        (* Warnung Hand Ein *)
		ayWarningReporter[3].proPrio	:= 3;    
		ayWarningReporter[3].proHandLokal :=    xIsHandOn;
		ayWarningReporter[3].metReport(			xSetReportIn					:= xIsHandOn,
												iReportID						:= 3,
												enReportTypeIn					:= CtaAppReport.enReportType.Warning,  
												enReportAcknowledgeTypeIn   	:= CtaAppReport.enReportAcknowledgeType.Auto,
												tDelay							:= T#0S, 
												ITF_BMK_IN						:= THIS^,			              
												pstReportTextListIn				:= ADR(GlobalKonstant.stReportTextListWarning),
												stOptionalReportText		    := '',   
												iRetryTilReportLock 		    := 0, 
												xResetCount         		    := FALSE,  
												tReset						    := T#0S);   
 
        (* Warnung Handmodul Actuator *)
		ayWarningReporter[4].proPrio	:= 4;    
		ayWarningReporter[4].proHandLokal :=    xActuatorHand;
		ayWarningReporter[4].metReport(			xSetReportIn					:= xActuatorHand,
												iReportID						:= 4,
												enReportTypeIn					:= CtaAppReport.enReportType.Warning,  
												enReportAcknowledgeTypeIn   	:= CtaAppReport.enReportAcknowledgeType.Auto,
												tDelay							:= T#0S, 
												ITF_BMK_IN						:= THIS^,			              
												pstReportTextListIn				:= ADR(GlobalKonstant.stReportTextListWarning),
												stOptionalReportText		    := '',   
												iRetryTilReportLock 		    := 0, 
												xResetCount         		    := FALSE,  
												tReset						    := T#0S);                                                   
(* Sync Reports *)                                         
FOR difor := LOWER_BOUND(ayErrorReporter,1) TO UPPER_BOUND(ayErrorReporter,1) DO
	fbReportManager.metSyncReporter(ayErrorReporter[difor]);	
END_FOR;
FOR difor := LOWER_BOUND(ayWarningReporter,1) TO UPPER_BOUND(ayWarningReporter,1) DO
	fbReportManager.metSyncReporter(ayWarningReporter[difor]);	
END_FOR;
                                                                             
_xIsError   := scEWI.iError <> 0;
_xIsWarning := scEWI.iWarning <> 0;
END_ACTION

{attribute 'monitoring' := 'variable'}
PROPERTY proAcknowlege : BOOL
GET
proAcknowlege :=NOT proIsError;
END_GET
END_PROPERTY

{attribute 'monitoring' := 'variable'}
PROPERTY proAvailable : BOOL
GET
proAvailable := proIsReady;
END_GET
END_PROPERTY

{attribute 'monitoring' := 'variable'}
PROPERTY proLockDown : BOOL
GET
proLockDown := proIsError;
END_GET
END_PROPERTY

END_FUNCTION_BLOCK

// 30 Program Organization Units/Abstracte Bausteine/fbSperrAntriebTabellenInfo
{attribute 'hide'} 
FUNCTION_BLOCK INTERNAL ABSTRACT fbSperrAntriebTabellenInfo EXTENDS CtaAppBmk.fbBMK IMPLEMENTS ITF_SPERRANTRIEB_TABELLE_INFO

PROPERTY proOnAuf : BOOL
GET
END_GET
END_PROPERTY

PROPERTY proStateSymbol : STRING
GET
END_GET
END_PROPERTY

PROPERTY proEnSymbol : STRING
GET
END_GET
END_PROPERTY

PROPERTY proIsOn : BOOL
GET
END_GET
END_PROPERTY

PROPERTY proIsOnY : REAL
GET
END_GET
END_PROPERTY

PROPERTY proOn : BOOL
GET
END_GET
END_PROPERTY

PROPERTY proOnY : REAL
GET
END_GET
END_PROPERTY

PROPERTY proOnZu : BOOL
GET
END_GET
END_PROPERTY

PROPERTY proRükIsClosed : BOOL
GET
END_GET
END_PROPERTY

PROPERTY proRükIsOpen : BOOL
GET
END_GET
END_PROPERTY

END_FUNCTION_BLOCK

// 21 Interface/ITF_SPERRANTRIEB_TABELLE_INFO
INTERFACE INTERNAL ITF_SPERRANTRIEB_TABELLE_INFO EXTENDS CtaAppBmk.ITF_BMK

PROPERTY proRükIsOpen : BOOL
GET
END_GET
END_PROPERTY

PROPERTY proRükIsClosed : BOOL
GET
END_GET
END_PROPERTY

PROPERTY INTERNAL proStateSymbol : STRING
GET
END_GET
END_PROPERTY

PROPERTY INTERNAL proEnSymbol : STRING
GET
END_GET
END_PROPERTY

PROPERTY proOnZu : BOOL
GET
END_GET
END_PROPERTY

PROPERTY proIsOnY : REAL
GET
END_GET
END_PROPERTY

PROPERTY proOnAuf : BOOL
GET
END_GET
END_PROPERTY

PROPERTY proOnY : REAL
GET
END_GET
END_PROPERTY

END_INTERFACE

// 21 Interface/ITF_SPERRANTRIEB
INTERFACE ITF_SPERRANTRIEB EXTENDS ITF_SPERRANTRIEB_TABELLE_INFO, CtaAppModbusSpezifikation.ITF_MODBUS_SPEZIFIKATION

PROPERTY proAuto : BOOL
GET
END_GET
SET
END_SET
END_PROPERTY

PROPERTY proHandOff : BOOL
GET
END_GET
SET
END_SET
END_PROPERTY

PROPERTY proHandOn : BOOL
GET
END_GET
SET
END_SET
END_PROPERTY

PROPERTY proIsRegulatet : BOOL
GET
END_GET
END_PROPERTY

PROPERTY proIsError : BOOL
GET
END_GET
END_PROPERTY

PROPERTY proIsWarning : BOOL
GET
END_GET
END_PROPERTY

PROPERTY proIsEnabled : BOOL
GET
END_GET
END_PROPERTY

PROPERTY proIsHandOnOrOff : BOOL
GET
END_GET
END_PROPERTY

PROPERTY proIsReady : BOOL
GET
END_GET
END_PROPERTY

PROPERTY proHardWareHandModulAktive : BOOL
GET
END_GET
END_PROPERTY

PROPERTY proRevisionSwitchOk : BOOL
GET
END_GET
END_PROPERTY

PROPERTY proHandManualClose : BOOL
SET
END_SET
GET
END_GET
END_PROPERTY

PROPERTY proEn : BOOL
SET
END_SET
GET
END_GET
END_PROPERTY

PROPERTY proGetDI_RükIsOpen : BOOL
GET
END_GET
END_PROPERTY

PROPERTY proNotShowDI_RükIsOpen : BOOL
GET
END_GET
END_PROPERTY

PROPERTY proIsOpen_ITF : CtaSysIO.ITF_IO
GET
END_GET
END_PROPERTY

PROPERTY INTERNAL proGetDI_ActuatorHand : BOOL
GET
END_GET
END_PROPERTY

PROPERTY proNotShowDI_ActuatorHand : BOOL
GET
END_GET
END_PROPERTY

PROPERTY proHandModul_ITF : CtaSysIO.ITF_IO
GET
END_GET
END_PROPERTY

PROPERTY INTERNAL proGetDI_ActuatorFuseOk : BOOL
GET
END_GET
END_PROPERTY

PROPERTY proNotShowDI_ActuatorFuseOk : BOOL
GET
END_GET
END_PROPERTY

PROPERTY proActuatorFuse_ITF : CtaSysIO.ITF_IO
GET
END_GET
END_PROPERTY

PROPERTY INTERNAL proGetDI_IsReady : BOOL
GET
END_GET
END_PROPERTY

PROPERTY proNotShowDI_Ready : BOOL
GET
END_GET
END_PROPERTY

PROPERTY proActuatorReady_ITF : CtaSysIO.ITF_IO
GET
END_GET
END_PROPERTY

PROPERTY INTERNAL proGetDI_FuseOK : BOOL
GET
END_GET
END_PROPERTY

PROPERTY proNotShowDI_FuseOk : BOOL
GET
END_GET
END_PROPERTY

PROPERTY proFuse_ITF : CtaSysIO.ITF_IO
GET
END_GET
END_PROPERTY

PROPERTY INTERNAL proGetDI_RevisionSwitchOK : BOOL
GET
END_GET
END_PROPERTY

PROPERTY proNotShowDI_RevisionSwitchOk : BOOL
GET
END_GET
END_PROPERTY

PROPERTY proRevisionSwitch_ITF : CtaSysIO.ITF_IO
GET
END_GET
END_PROPERTY

PROPERTY proNotShowAI_ActualPosition : BOOL
GET
END_GET
END_PROPERTY

PROPERTY proGetAI_ActualPosition : REAL
GET
END_GET
END_PROPERTY

PROPERTY proActualPosition_ITF : CtaSysIO.ITF_IO
GET
END_GET
END_PROPERTY

PROPERTY proGetDI_RükIsClosed : BOOL
GET
END_GET
END_PROPERTY

PROPERTY proNotShowDI_RükIsClosed : BOOL
GET
END_GET
END_PROPERTY

PROPERTY proIsClosed_ITF : CtaSysIO.ITF_IO
GET
END_GET
END_PROPERTY

PROPERTY proOnY_ITF : CtaSysIO.ITF_IO
GET
END_GET
END_PROPERTY

PROPERTY proOnOpen_ITF : CtaSysIO.ITF_IO
GET
END_GET
END_PROPERTY

PROPERTY proOnClose_ITF : CtaSysIO.ITF_IO
GET
END_GET
END_PROPERTY

PROPERTY INTERNAL proAnzWarning : INT
GET
END_GET
END_PROPERTY

PROPERTY INTERNAL proITF_REPORTMANAGER : CtaAppReport.ITF_REPORTMANAGER
GET
END_GET
END_PROPERTY

PROPERTY INTERNAL proAnzInfo : INT
GET
END_GET
END_PROPERTY

PROPERTY INTERNAL proAnzError : INT
GET
END_GET
END_PROPERTY

PROPERTY INTERNAL proModbusTest : BOOL
SET
END_SET
GET
END_GET
END_PROPERTY

PROPERTY proModbusStateWord : REFERENCE TO ARRAY[0..3] OF WORD
GET
END_GET
END_PROPERTY

PROPERTY proModbusControllWord : REFERENCE TO ARRAY[0..3] OF WORD
GET
END_GET
END_PROPERTY

PROPERTY proConfigError : BOOL
GET
END_GET
END_PROPERTY

PROPERTY p_scBase_fbxEnable : CtaSysConfig.ITF_DATATYPE;
GET
END_GET
END_PROPERTY

PROPERTY p_scBase_fbxControllMb : CtaSysConfig.ITF_DATATYPE;
GET
END_GET
END_PROPERTY

PROPERTY p_scBase_fbxInvertiert : CtaSysConfig.ITF_DATATYPE;
GET
END_GET
END_PROPERTY

PROPERTY p_scBase_fbtSettingTime : CtaSysConfig.ITF_DATATYPE;
GET
END_GET
END_PROPERTY

PROPERTY p_scFuse_fbxEnable : CtaSysConfig.ITF_DATATYPE;
GET
END_GET
END_PROPERTY

PROPERTY p_scFuse_fbxInputMb : CtaSysConfig.ITF_DATATYPE;
GET
END_GET
END_PROPERTY

PROPERTY p_scFuse_fbxDoesAlarm : CtaSysConfig.ITF_DATATYPE;
GET
END_GET
END_PROPERTY

PROPERTY p_scActuatorFuse_fbxEnable : CtaSysConfig.ITF_DATATYPE;
GET
END_GET
END_PROPERTY

PROPERTY p_scActuatorFuse_fbxInputMb : CtaSysConfig.ITF_DATATYPE;
GET
END_GET
END_PROPERTY

PROPERTY p_scActuatorFuse_fbxDoesAlarm : CtaSysConfig.ITF_DATATYPE;
GET
END_GET
END_PROPERTY

PROPERTY p_scInSperrAtRevisionSwitch_fbxEnable : CtaSysConfig.ITF_DATATYPE;
GET
END_GET
END_PROPERTY

PROPERTY p_scInSperrAtRevisionSwitch_fbxInputMb : CtaSysConfig.ITF_DATATYPE;
GET
END_GET
END_PROPERTY

PROPERTY p_scInSperrAtReady_fbxEnable : CtaSysConfig.ITF_DATATYPE;
GET
END_GET
END_PROPERTY

PROPERTY p_scInSperrAtReady_fbxInputMb : CtaSysConfig.ITF_DATATYPE;
GET
END_GET
END_PROPERTY

PROPERTY p_scInSperrAtHand_fbxEnable : CtaSysConfig.ITF_DATATYPE;
GET
END_GET
END_PROPERTY

PROPERTY p_scInSperrAtHand_fbxInputMb : CtaSysConfig.ITF_DATATYPE;
GET
END_GET
END_PROPERTY

PROPERTY p_scInSperrAtRükClosed_fbxEnable : CtaSysConfig.ITF_DATATYPE;
GET
END_GET
END_PROPERTY

PROPERTY p_scInSperrAtRükClosed_fbxInputMb : CtaSysConfig.ITF_DATATYPE;
GET
END_GET
END_PROPERTY

PROPERTY p_scInSperrAtRükClosed_fbxDoesAlarm : CtaSysConfig.ITF_DATATYPE;
GET
END_GET
END_PROPERTY

PROPERTY p_scInSperrAtRükClosed_fbtDelayStart : CtaSysConfig.ITF_DATATYPE;
GET
END_GET
END_PROPERTY

PROPERTY p_scInSperrAtRükClosed_fbtDelayRun : CtaSysConfig.ITF_DATATYPE;
GET
END_GET
END_PROPERTY

PROPERTY p_scInSperrAtRükClosed_fbiTypeOfAck : CtaSysConfig.ITF_DATATYPE;
GET
END_GET
END_PROPERTY

PROPERTY p_scInSperrAtRükClosed_fbiMaxErrorRetryAllowed : CtaSysConfig.ITF_DATATYPE;
GET
END_GET
END_PROPERTY

PROPERTY p_scInSperrAtRükOpen_fbxEnable : CtaSysConfig.ITF_DATATYPE;
GET
END_GET
END_PROPERTY

PROPERTY p_scInSperrAtRükOpen_fbxInputMb : CtaSysConfig.ITF_DATATYPE;
GET
END_GET
END_PROPERTY

PROPERTY p_scInSperrAtRükOpen_fbxDoesAlarm : CtaSysConfig.ITF_DATATYPE;
GET
END_GET
END_PROPERTY

PROPERTY p_scInSperrAtRükOpen_fbtDelayStart : CtaSysConfig.ITF_DATATYPE;
GET
END_GET
END_PROPERTY

PROPERTY p_scInSperrAtRükOpen_fbtDelayRun : CtaSysConfig.ITF_DATATYPE;
GET
END_GET
END_PROPERTY

PROPERTY p_scInSperrAtRükOpen_fbiTypeOfAck : CtaSysConfig.ITF_DATATYPE;
GET
END_GET
END_PROPERTY

PROPERTY p_scInSperrAtRükOpen_fbiMaxErrorRetryAllowed : CtaSysConfig.ITF_DATATYPE;
GET
END_GET
END_PROPERTY

PROPERTY p_scInSperrAtActualPosition_fbxEnable : CtaSysConfig.ITF_DATATYPE;
GET
END_GET
END_PROPERTY

PROPERTY p_scInSperrAtActualPosition_fbxInputMb : CtaSysConfig.ITF_DATATYPE;
GET
END_GET
END_PROPERTY

PROPERTY p_scInSperrAtActualPosition_fbxDoesAlarm : CtaSysConfig.ITF_DATATYPE;
GET
END_GET
END_PROPERTY

PROPERTY p_scInSperrAtActualPosition_fbrMaxDiff : CtaSysConfig.ITF_DATATYPE;
GET
END_GET
END_PROPERTY

PROPERTY p_scInSperrAtActualPosition_fbtDelayStart : CtaSysConfig.ITF_DATATYPE;
GET
END_GET
END_PROPERTY

PROPERTY p_scInSperrAtActualPosition_fbtDelayRun : CtaSysConfig.ITF_DATATYPE;
GET
END_GET
END_PROPERTY

PROPERTY p_scInSperrAtActualPosition_fbiTypeOfAck : CtaSysConfig.ITF_DATATYPE;
GET
END_GET
END_PROPERTY

PROPERTY p_scInSperrAtActualPosition_fbiMaxErrorRetryAllowed : CtaSysConfig.ITF_DATATYPE;
GET
END_GET
END_PROPERTY

PROPERTY p_scInfluxDb_fbxEnable : CtaSysConfig.ITF_DATATYPE;
GET
END_GET
END_PROPERTY

PROPERTY p_scManual_fbxAlowManualOn : CtaSysConfig.ITF_DATATYPE;
GET
END_GET
END_PROPERTY

PROPERTY p_scManual_fbuiManualState : CtaSysConfig.ITF_DATATYPE;
GET
END_GET
END_PROPERTY

PROPERTY p_scManual_fbuiSchaltBefehl : CtaSysConfig.ITF_DATATYPE;
GET
END_GET
END_PROPERTY

PROPERTY proHandManualOpen : BOOL
GET
END_GET
SET
END_SET
END_PROPERTY

PROPERTY proIsInverted : BOOL
GET
END_GET
END_PROPERTY

PROPERTY proKlappenStatus : enKlappenStatus
GET
END_GET
END_PROPERTY

PROPERTY proValveIcon : UINT
GET
END_GET
SET
END_SET
END_PROPERTY

{attribute 'monitoring' := 'variable'}
PROPERTY proAcknowlege : BOOL
GET
END_GET
END_PROPERTY

{attribute 'monitoring' := 'variable'}
PROPERTY proAvailable : BOOL
GET
END_GET
END_PROPERTY

{attribute 'monitoring' := 'variable'}
PROPERTY proLockDown : BOOL
GET
END_GET
END_PROPERTY

PROPERTY proOn : BOOL
GET
END_GET
END_PROPERTY

END_INTERFACE

// 30 Program Organization Units/fbSperrAntrieb_Collector
FUNCTION_BLOCK fbSperrAntrieb_Collector IMPLEMENTS ITF_SPERRAT_COLLECTOR
VAR_INPUT
END_VAR
VAR_OUTPUT
END_VAR
VAR
    aySperrAT_INTERFACE          : ARRAY[1..Parameter.iMaxSperrAntrieb] OF ITF_SPERRANTRIEB;   
    aySperrAT_INTERFACE_SORTET   : ARRAY[1..Parameter.iMaxSperrAntrieb] OF ITF_SPERRANTRIEB; 
    xIsSortet               : BOOL;
    diNext                  : DINT    := 1;
    diMin                   : DINT    := 1;
    diMax                   : DINT;
    diMaxSort               : DINT;
    xError                  : BOOL;
    xBufferError            : BOOL;
    diMissedBuffer          : DINT;
END_VAR

METHOD metRegistry : DINT
VAR_INPUT
    ITF_AT_IN   :   ITF_SPERRANTRIEB;
END_VAR
VAR
    diArrayPos  :   DINT;
    diCount     :   DINT;
END_VAR
IF ITF_AT_IN <> 0 THEN
    diArrayPos := __XADD(ADR(diNext),1);
    IF diArrayPos <= Parameter.iMaxSperrAntrieb AND diArrayPos >= 1 THEN
        IF __QUERYINTERFACE(ITF_AT_IN,aySperrAT_INTERFACE[diArrayPos]) THEN
            metRegistry             := diArrayPos;
            GVL_SperrAntrieb.xValidData       := TRUE;
            diCount    := __XADD(ADR(diMax),1);
        END_IF;
    ELSE
        IF diArrayPos > Parameter.iMaxSperrAntrieb THEN
            xBufferError := TRUE;
            diMissedBuffer := diArrayPos - Parameter.iMaxSperrAntrieb;
		END_IF;
        xError      := TRUE; 
        metRegistry := 0;
    END_IF;   
ELSE
    xError := TRUE; 
    metRegistry := 0;
END_IF;
END_METHOD

METHOD metSortArray
VAR_INPUT
    stSearch    :   STRING;
    uiSort      :   UINT;
END_VAR
VAR
    diFor1      :   DINT;
    diFor2      :   DINT;
    diFill      :   DINT;
    ITF_AT_Temp :   ITF_SPERRANTRIEB;    
    iBigger     :   INT;
END_VAR
IF stSearch <> '' THEN
    diMaxSort   := 0;
    diFill      := LOWER_BOUND(aySperrAT_INTERFACE,1); 
    FOR diFor1 := LOWER_BOUND(aySperrAT_INTERFACE,1) TO UPPER_BOUND(aySperrAT_INTERFACE,1) DO
        IF aySperrAT_INTERFACE[diFor1] <> 0 THEN
            IF FIND(aySperrAT_INTERFACE[diFor1].proGetBMK,stSearch) <> 0 OR FIND(aySperrAT_INTERFACE[diFor1].proGetVendorDesignation,stSearch) <> 0 THEN
                aySperrAT_INTERFACE_SORTET[diFill] := aySperrAT_INTERFACE[diFor1];
                diFill      := diFill + 1; 
                diMaxSort   := diFill -1; 
            END_IF;
        END_IF;
	END_FOR;
ELSE
    aySperrAT_INTERFACE_SORTET := aySperrAT_INTERFACE;
    diMaxSort := diMax;
END_IF; 
// 1 = Sort BMK
IF uiSort = 1 THEN
    FOR diFor1 := LOWER_BOUND(aySperrAT_INTERFACE_SORTET,1) TO diMaxSort DO 
        FOR diFor2 := LOWER_BOUND(aySperrAT_INTERFACE_SORTET,1) TO diMaxSort -1 DO 
            IF aySperrAT_INTERFACE_SORTET[diFor2] <> 0 AND aySperrAT_INTERFACE_SORTET[diFor2 + 1] <> 0 THEN
                IF LEN(aySperrAT_INTERFACE_SORTET[diFor2].proGetBMK) > LEN(aySperrAT_INTERFACE_SORTET[diFor2 + 1].proGetBMK) THEN
                    ITF_AT_Temp                         := aySperrAT_INTERFACE_SORTET[diFor2];
                    aySperrAT_INTERFACE_SORTET[diFor2]       := aySperrAT_INTERFACE_SORTET[diFor2 + 1];
                    aySperrAT_INTERFACE_SORTET[diFor2 + 1]   := ITF_AT_Temp; 
                ELSIF LEN(aySperrAT_INTERFACE_SORTET[diFor2].proGetBMK) = LEN(aySperrAT_INTERFACE_SORTET[diFor2 + 1].proGetBMK) THEN
                    iBigger := fcGetBigerStringValue(aySperrAT_INTERFACE_SORTET[diFor2].proGetBMK,aySperrAT_INTERFACE_SORTET[diFor2 + 1].proGetBMK);
                    IF iBigger = 1 THEN
                        ITF_AT_Temp                         := aySperrAT_INTERFACE_SORTET[diFor2];
                        aySperrAT_INTERFACE_SORTET[diFor2]       := aySperrAT_INTERFACE_SORTET[diFor2 + 1];
                        aySperrAT_INTERFACE_SORTET[diFor2 + 1]   := ITF_AT_Temp;                                                
					END_IF;
				END_IF;
            END_IF;       
        END_FOR;      
    END_FOR;     
// 2 = Sort Vendor Name    
ELSIF uiSort = 2 THEN
    FOR diFor1 := LOWER_BOUND(aySperrAT_INTERFACE_SORTET,1) TO diMaxSort DO 
        FOR diFor2 := LOWER_BOUND(aySperrAT_INTERFACE_SORTET,1) TO diMaxSort -1 DO 
            IF aySperrAT_INTERFACE_SORTET[diFor2] <> 0 AND aySperrAT_INTERFACE_SORTET[diFor2 + 1] <> 0 THEN
                iBigger := fcGetBigerStringValue(aySperrAT_INTERFACE_SORTET[diFor2].proGetVendorDesignation,aySperrAT_INTERFACE_SORTET[diFor2 + 1].proGetVendorDesignation);
                IF iBigger = 1 THEN
                    ITF_AT_Temp                         := aySperrAT_INTERFACE_SORTET[diFor2];
                    aySperrAT_INTERFACE_SORTET[diFor2]       := aySperrAT_INTERFACE_SORTET[diFor2 + 1];
                    aySperrAT_INTERFACE_SORTET[diFor2 + 1]   := ITF_AT_Temp;                                            
                END_IF;
            END_IF;       
        END_FOR;      
    END_FOR;
// 3 & 4 = Sort State  
ELSIF uiSort = 3 OR uiSort = 4 THEN
    FOR diFor1 := LOWER_BOUND(aySperrAT_INTERFACE_SORTET,1) TO diMaxSort DO 
        FOR diFor2 := LOWER_BOUND(aySperrAT_INTERFACE_SORTET,1) TO diMaxSort -1 DO 
            IF aySperrAT_INTERFACE_SORTET[diFor2] <> 0 AND aySperrAT_INTERFACE_SORTET[diFor2 + 1] <> 0 THEN
                IF aySperrAT_INTERFACE_SORTET[diFor2].proIsError < aySperrAT_INTERFACE_SORTET[diFor2 + 1].proIsError THEN
                    ITF_AT_Temp                         := aySperrAT_INTERFACE_SORTET[diFor2];
                    aySperrAT_INTERFACE_SORTET[diFor2]       := aySperrAT_INTERFACE_SORTET[diFor2 + 1];
                    aySperrAT_INTERFACE_SORTET[diFor2 + 1]   := ITF_AT_Temp;    
                ELSIF NOT aySperrAT_INTERFACE_SORTET[diFor2].proIsError THEN
                    IF aySperrAT_INTERFACE_SORTET[diFor2].proIsWarning < aySperrAT_INTERFACE_SORTET[diFor2 + 1].proIsWarning THEN
                        ITF_AT_Temp                         := aySperrAT_INTERFACE_SORTET[diFor2];
                        aySperrAT_INTERFACE_SORTET[diFor2]       := aySperrAT_INTERFACE_SORTET[diFor2 + 1];
                        aySperrAT_INTERFACE_SORTET[diFor2 + 1]   := ITF_AT_Temp;    
                    ELSIF aySperrAT_INTERFACE_SORTET[diFor2].proIsEnabled < aySperrAT_INTERFACE_SORTET[diFor2 + 1].proIsEnabled THEN
                        ITF_AT_Temp                         := aySperrAT_INTERFACE_SORTET[diFor2];
                        aySperrAT_INTERFACE_SORTET[diFor2]       := aySperrAT_INTERFACE_SORTET[diFor2 + 1];
                        aySperrAT_INTERFACE_SORTET[diFor2 + 1]   := ITF_AT_Temp; 
                    ELSIF aySperrAT_INTERFACE_SORTET[diFor2].proIsWarning AND aySperrAT_INTERFACE_SORTET[diFor2 + 1].proIsWarning THEN
                        IF aySperrAT_INTERFACE_SORTET[diFor2].proRevisionSwitchOk > aySperrAT_INTERFACE_SORTET[diFor2 + 1].proRevisionSwitchOk THEN         
                            ITF_AT_Temp                         := aySperrAT_INTERFACE_SORTET[diFor2];
                            aySperrAT_INTERFACE_SORTET[diFor2]       := aySperrAT_INTERFACE_SORTET[diFor2 + 1];
                            aySperrAT_INTERFACE_SORTET[diFor2 + 1]   := ITF_AT_Temp; 
                        END_IF;       
                    END_IF;                                                       
                END_IF;
            END_IF;       
        END_FOR;      
    END_FOR;    
// 5 = Sort Befehlt AUF  
ELSIF uiSort = 5 THEN
    FOR diFor1 := LOWER_BOUND(aySperrAT_INTERFACE_SORTET,1) TO diMaxSort DO 
        FOR diFor2 := LOWER_BOUND(aySperrAT_INTERFACE_SORTET,1) TO diMaxSort -1 DO 
            IF aySperrAT_INTERFACE_SORTET[diFor2] <> 0 AND aySperrAT_INTERFACE_SORTET[diFor2 + 1] <> 0 THEN
                IF aySperrAT_INTERFACE_SORTET[diFor2].proOnAuf < aySperrAT_INTERFACE_SORTET[diFor2 + 1].proOnAuf THEN
                    ITF_AT_Temp                         := aySperrAT_INTERFACE_SORTET[diFor2];
                    aySperrAT_INTERFACE_SORTET[diFor2]       := aySperrAT_INTERFACE_SORTET[diFor2 + 1];
                    aySperrAT_INTERFACE_SORTET[diFor2 + 1]   := ITF_AT_Temp;                                            
                END_IF;
            END_IF;       
        END_FOR;      
    END_FOR; 
// 6 = Sort Befehl ZU   
ELSIF uiSort = 6 THEN
    FOR diFor1 := LOWER_BOUND(aySperrAT_INTERFACE_SORTET,1) TO diMaxSort DO 
        FOR diFor2 := LOWER_BOUND(aySperrAT_INTERFACE_SORTET,1) TO diMaxSort -1 DO 
            IF aySperrAT_INTERFACE_SORTET[diFor2] <> 0 AND aySperrAT_INTERFACE_SORTET[diFor2 + 1] <> 0 THEN
                IF aySperrAT_INTERFACE_SORTET[diFor2].proOnZu < aySperrAT_INTERFACE_SORTET[diFor2 + 1].proOnZu THEN
                    ITF_AT_Temp                         := aySperrAT_INTERFACE_SORTET[diFor2];
                    aySperrAT_INTERFACE_SORTET[diFor2]       := aySperrAT_INTERFACE_SORTET[diFor2 + 1];
                    aySperrAT_INTERFACE_SORTET[diFor2 + 1]   := ITF_AT_Temp;                                            
                END_IF;
            END_IF;       
        END_FOR;      
    END_FOR;   
// 7 = Sort Stellwert Y    
ELSIF uiSort = 7 THEN
    FOR diFor1 := LOWER_BOUND(aySperrAT_INTERFACE_SORTET,1) TO diMaxSort DO 
        FOR diFor2 := LOWER_BOUND(aySperrAT_INTERFACE_SORTET,1) TO diMaxSort -1 DO 
            IF aySperrAT_INTERFACE_SORTET[diFor2] <> 0 AND aySperrAT_INTERFACE_SORTET[diFor2 + 1] <> 0 THEN
                IF aySperrAT_INTERFACE_SORTET[diFor2].proOnY < aySperrAT_INTERFACE_SORTET[diFor2 + 1].proOnY THEN
                    ITF_AT_Temp                         := aySperrAT_INTERFACE_SORTET[diFor2];
                    aySperrAT_INTERFACE_SORTET[diFor2]       := aySperrAT_INTERFACE_SORTET[diFor2 + 1];
                    aySperrAT_INTERFACE_SORTET[diFor2 + 1]   := ITF_AT_Temp;                                            
                END_IF;
            END_IF;       
        END_FOR;      
    END_FOR;   
ELSE
    uiSort := 0;     
END_IF; 
IF uiSort = 0 AND stSearch = '' THEN
    xIsSortet := FALSE;  
ELSE
    xIsSortet := TRUE;  
END_IF
END_METHOD

PROPERTY proMin : INT
GET
proMin := 1;
END_GET
END_PROPERTY

PROPERTY proMax : UINT
GET
IF xIsSortet THEN
    proMax := LIMIT(0,TO_UINT(diMaxSort),65535);    
ELSE
    proMax := LIMIT(0,TO_UINT(diMax),65535);    
END_IF
END_GET
END_PROPERTY

PROPERTY proaySperrAntriebTabelle : ARRAY[1..Parameter.iMaxSperrAntrieb] OF ITF_SPERRANTRIEB_TABELLE_INFO
GET
VAR
    diFor   :   DINT;
END_VAR
IF xIsSortet THEN
    FOR diFor := LOWER_BOUND(proaySperrAntriebTabelle,1) TO UPPER_BOUND(proaySperrAntriebTabelle,1) DO
        __QUERYINTERFACE(aySperrAT_INTERFACE_SORTET[diFor],proaySperrAntriebTabelle[diFor]);   
	END_FOR
ELSE
    FOR diFor := LOWER_BOUND(proaySperrAntriebTabelle,1) TO UPPER_BOUND(proaySperrAntriebTabelle,1) DO
        __QUERYINTERFACE(aySperrAT_INTERFACE[diFor],proaySperrAntriebTabelle[diFor]);   
	END_FOR
END_IF;
END_GET
END_PROPERTY

PROPERTY proMissedBuffer : DINT
GET
proMissedBuffer := diMissedBuffer;
END_GET
END_PROPERTY

PROPERTY proBufferError : BOOL
GET
proBufferError := xBufferError;
END_GET
END_PROPERTY

PROPERTY proaySperrAntrieb : ARRAY[1..Parameter.iMaxSperrAntrieb] OF ITF_SPERRANTRIEB
GET
VAR
    diFor   :   DINT;
END_VAR
IF xIsSortet THEN
    proaySperrAntrieb := aySperrAT_INTERFACE_SORTET;
ELSE
    proaySperrAntrieb := aySperrAT_INTERFACE;
END_IF;
END_GET
END_PROPERTY

METHOD metGetStellAntriebITF : ITF_SPERRANTRIEB
VAR_INPUT
    iPos    :   INT;
END_VAR
IF TO_DINT(iPos) >= LOWER_BOUND(aySperrAT_INTERFACE,1) AND TO_DINT(iPos) <= UPPER_BOUND(aySperrAT_INTERFACE,1) THEN
    IF xIsSortet THEN
        metGetStellAntriebITF := aySperrAT_INTERFACE_SORTET[iPos];       
    ELSE
        metGetStellAntriebITF := aySperrAT_INTERFACE[iPos];       
	END_IF   
END_IF
END_METHOD

END_FUNCTION_BLOCK

// 21 Interface/ITF_SPERRAT_COLLECTOR
INTERFACE ITF_SPERRAT_COLLECTOR

METHOD metSortArray
VAR_INPUT
    stSearch    :   STRING;
    uiSort      :   UINT;
END_VAR
END_METHOD

PROPERTY proaySperrAntriebTabelle : ARRAY[1..Parameter.iMaxSperrAntrieb] OF ITF_SPERRANTRIEB_TABELLE_INFO
GET
END_GET
END_PROPERTY

PROPERTY proMax : UINT
GET
END_GET
END_PROPERTY

PROPERTY proMin : INT
GET
END_GET
END_PROPERTY

PROPERTY proBufferError : BOOL
GET
END_GET
END_PROPERTY

PROPERTY proMissedBuffer : DINT
GET
END_GET
END_PROPERTY

METHOD metGetStellAntriebITF : ITF_SPERRANTRIEB
VAR_INPUT
    iPos    :   INT;
END_VAR
END_METHOD

END_INTERFACE

// 30 Program Organization Units/fcGetBigerStringValue
FUNCTION fcGetBigerStringValue : INT
VAR_INPUT
    st1     :   STRING(255);
    st2     :   STRING(255);
END_VAR
VAR
    diFor: DINT;
    diMax: DINT;
END_VAR

IF LEN(st1) > LEN(st2) THEN
    diMax := LEN(st2); 
    fcGetBigerStringValue := 1;
ELSIF LEN(st1) < LEN(st2) THEN
    diMax := LEN(st1);
    fcGetBigerStringValue := 2;     
ELSE
    diMax := LEN(st1);    
END_IF;
FOR diFor := 0 TO  diMax DO
    IF st1[diFor] > st2[diFor] THEN
        fcGetBigerStringValue := 1;  
        EXIT; 
    ELSIF st1[diFor] < st2[diFor] THEN
        fcGetBigerStringValue := 2;  
        EXIT;
    END_IF;
END_FOR;

END_FUNCTION

// 30 Program Organization Units/fcCheckQuerryReturnIcon
FUNCTION fcCheckQuerryReturnIcon : BOOL
VAR_INPUT
	_ITF_In			:	ITF_SPERRANTRIEB;
	_uiIconNr_In	:	UINT;
END_VAR

IF __QUERYINTERFACE(_ITF_In,_ITF_In) THEN	
	fcCheckQuerryReturnIcon := TRUE;	
	_ITF_In.proValveIcon := _uiIconNr_In;
ELSE
	fcCheckQuerryReturnIcon := FALSE;	
END_IF

END_FUNCTION

// 40 Visualizations/COLLECTOR/SperrAntrieb_Collector
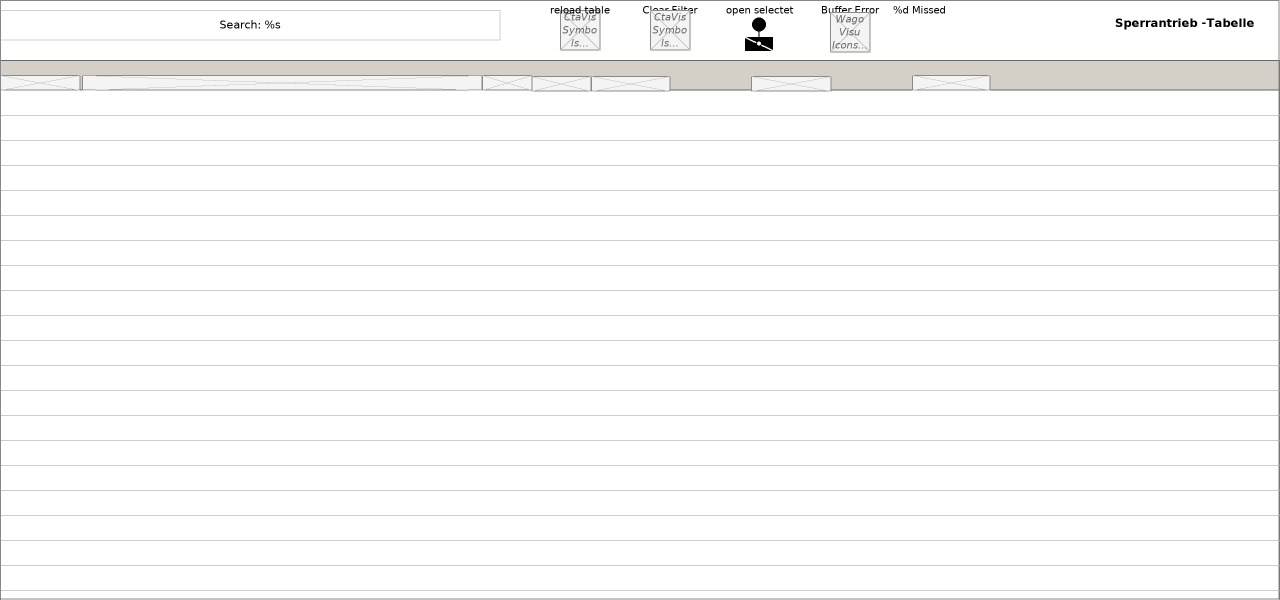
VISUALIZATION SperrAntrieb_Collector  // 1280x600
    Frame (0,0 1280x600), invisible if: NOT GVL_SperrAntrieb.xValidData
        shows SperrAntrieb_Collector_TEMP(aySperrAntriebTabellenInfo := GVL_SperrAntrieb.fbSperrAntrieb_Collector.proaySperrAntriebTabelle, uiMax := GVL_SperrAntrieb.fbSperrAntrieb_Collector.proMax, ITF_SPERRAT_COLLECTOR := GVL_SperrAntrieb.fbSperrAntrieb_Collector)
END_VISUALIZATION

// 40 Visualizations/COLLECTOR/Help Funktionen/SelSort
VISUALIZATION SelSort  // 15x30
VAR_IN_OUT
	uiSel               :   UINT;
END_VAR
VAR_INPUT
    stSearch            :   STRING;    
    ITF_SPERRAT_COLLECTOR    : ITF_SPERRAT_COLLECTOR;
END_VAR
VAR_INPUT CONSTANT
    uiValue             :   UINT;
END_VAR
    Frame (0,15 15x15), invisible if: uiValue <> uiSel
        shows SortPfeil()
    Rectangle (0,0 15x30)
        OnMouseClick: execute {
            IF uiSel <> uiValue THEN
                uiSel   := uiValue;
            ELSE
                uiSel   := 0;
            END_IF
            ITF_SPERRAT_COLLECTOR.metSortArray(stSearch,uiSel);
        }
END_VISUALIZATION

// 40 Visualizations/COLLECTOR/SperrAntrieb_Collector_TEMP
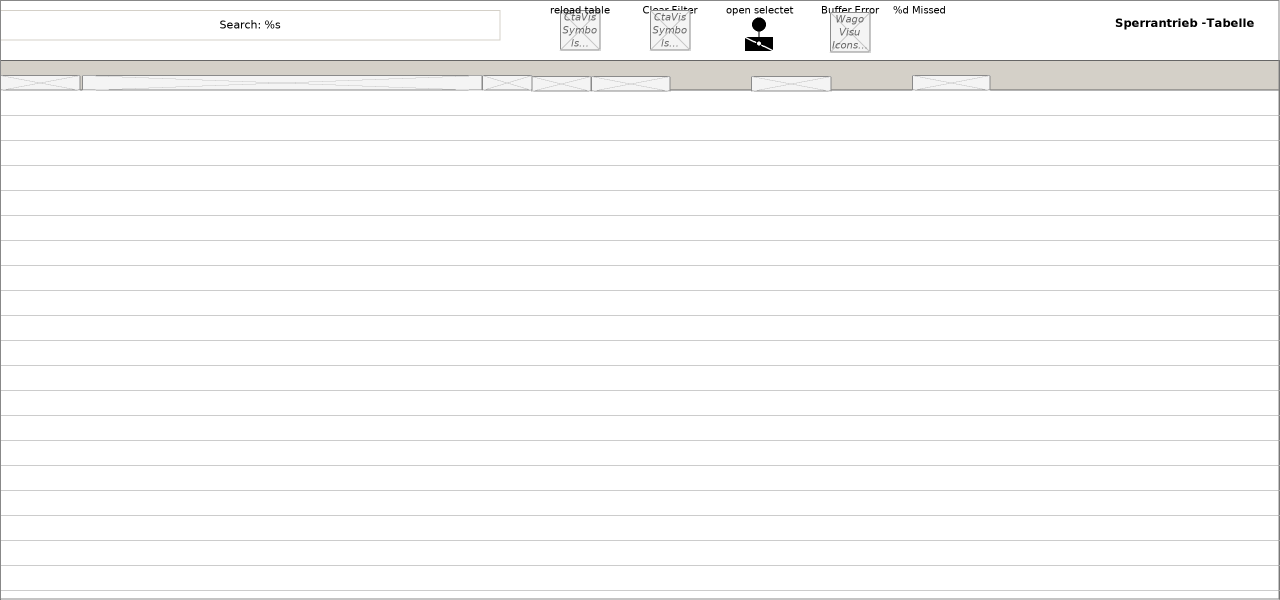
VISUALIZATION SperrAntrieb_Collector_TEMP  // 1280x600
VAR_INPUT
	aySperrAntriebTabellenInfo  	: 	ARRAY[1..Parameter.iMaxSperrAntrieb] OF ITF_SPERRANTRIEB_TABELLE_INFO;
    uiMax                   		: 	UINT;
    ITF_SPERRAT_COLLECTOR        	:	ITF_SPERRAT_COLLECTOR;
END_VAR
VAR
    iZeile                  	:   INT;
    stSearch               		:   STRING;
    uiSort                  	:   UINT;
    xReadySearch           		:   BOOL;
END_VAR
    Table (0,60 1280x541), data array: aySperrAntriebTabellenInfo
        p1128707560: uiMax
        p1014161805: Parameter.iMaxSperrAntrieb - 1 + 1
        p1137915858: iZeile
        p3136911649: ayStellAntriebTabellenInfo[INDEX].proGetInstancePath
        p797552052: ayStellAntriebTabellenInfo[INDEX].proSetInstancePath
        p3854506369: aySperrAntriebTabellenInfo[INDEX].proGetBMK
        p1892666644: aySperrAntriebTabellenInfo[INDEX].proGetVendorDesignation
        p338671338: aySperrAntriebTabellenInfo[INDEX].proOnAuf
        p2170511999: aySperrAntriebTabellenInfo[INDEX].proOnY
        p1218418051: aySperrAntriebTabellenInfo[INDEX].proRükIsOpen
        p746581629: aySperrAntriebTabellenInfo[INDEX].proOnZu
        p3104783080: aySperrAntriebTabellenInfo[INDEX].proRükIsClosed
        p7306298: aySperrAntriebTabellenInfo[INDEX].proIsOnY
        p1933151965: aySperrAntriebTabellenInfo[INDEX].proStateSymbol
        p3863566920: aySperrAntriebTabellenInfo[INDEX].proGetObjectId
        p400160035: aySperrAntriebTabellenInfo[INDEX].proNoBmkInList
        p1265227338: aySperrAntriebTabellenInfo[INDEX].proGetInstancePath
        p3726181087: aySperrAntriebTabellenInfo[INDEX].proSetInstancePath
        p511219082: Vendor designation
        p4092479075: Enabled
        p2237128397: Open OUT
        p505689113: Open IN
        p1757482276: Close OUT
        p4088588272: Closed IN
        p2243050616: Y OUT
        p516019884: Y IN
        p1739542657: aySperrAntriebTabellenInfo[INDEX].proGetAKS
        p4242324053: aySperrAntriebTabellenInfo[INDEX].proGetCustomerDesignation
        p262371475: aySperrAntriebTabellenInfo[INDEX].proEnSymbol
    Textfield (0,10 500x30), "Search: %s", text variable: stSearch
        OnMouseClick: write the text variable via Default
        OnMouseClick: execute { xReadySearch := TRUE; }
    Image (560,10 40x40), invisible if: NOT xReadySearch, image: CtaVisSymbols.ImagePool.refresh_solo_black
        OnMouseClick: execute { ITF_SPERRAT_COLLECTOR.metSortArray(stSearch,uiSort); xReadySearch := FALSE; }
    Label (540,5 80x10), "reload table", invisible if: NOT xReadySearch
    Label (720,5 80x10), "open selectet", invisible if: TO_DINT(iZeile) < LOWER_BOUND(aySperrAntriebTabellenInfo,1) OR TO_DINT(iZeile) > UPPER_BOUND(aySperrAntriebTabellenInfo,1)
    Label (630,5 80x10), "Clear Filter", invisible if: stSearch = '' AND uiSort = 0
    Image (650,10 40x40), invisible if: stSearch = '' AND uiSort = 0, image: CtaVisSymbols.ImagePool.close_solo_black
        OnMouseClick: execute {
            stSearch := '';
            uiSort   := 0;
            ITF_SPERRAT_COLLECTOR.metSortArray(stSearch,uiSort);
            xReadySearch := FALSE;
        }
    Label (1095,8 180x30), "Sperrantrieb -Tabelle"
    Label (810,5 80x10), "Buffer Error", invisible if: NOT ITF_SPERRAT_COLLECTOR.proBufferError
    Image (830,12 40x40), invisible if: NOT ITF_SPERRAT_COLLECTOR.proBufferError, image: WagoVisuIcons.WagoIcons.4
    Textfield (890,5 100x10), "%d Missed", text variable: ITF_SPERRAT_COLLECTOR.proMissedBuffer, invisible if: NOT ITF_SPERRAT_COLLECTOR.proBufferError
    Frame (740,15 40x40), invisible if: TO_DINT(iZeile) < LOWER_BOUND(aySperrAntriebTabellenInfo,1) OR TO_DINT(iZeile) > UPPER_BOUND(aySperrAntriebTabellenInfo,1)
        shows SperrAntrieb_Icon_SperrAntrieb()
        OnMouseClick:  Dialog=SperrAntrieb_POPUP, Parameters={uiPopUpGruppe: 0, ITF_SPERRANTRIEBIN: ITF_SPERRAT_COLLECTOR.metGetStellAntriebITF(iZeile)}, OpenModal=True, OpenCentered=True
    Frame (912,60 78x30)
        shows SelSort(uiSel := uiSort, stSearch := stSearch, ITF_SPERRAT_COLLECTOR := ITF_SPERRAT_COLLECTOR, uiValue := 7)
    Frame (751,61 80x30)
        shows SelSort(uiSel := uiSort, stSearch := stSearch, ITF_SPERRAT_COLLECTOR := ITF_SPERRAT_COLLECTOR, uiValue := 6)
    Frame (591,61 79x30)
        shows SelSort(uiSel := uiSort, stSearch := stSearch, ITF_SPERRAT_COLLECTOR := ITF_SPERRAT_COLLECTOR, uiValue := 5)
    Frame (531,61 60x30)
        shows SelSort(uiSel := uiSort, stSearch := stSearch, ITF_SPERRAT_COLLECTOR := ITF_SPERRAT_COLLECTOR, uiValue := 4)
    Frame (482,60 50x30)
        shows SelSort(uiSel := uiSort, stSearch := stSearch, ITF_SPERRAT_COLLECTOR := ITF_SPERRAT_COLLECTOR, uiValue := 3)
    Frame (82,60 400x30)
        shows SelSort(uiSel := uiSort, stSearch := stSearch, ITF_SPERRAT_COLLECTOR := ITF_SPERRAT_COLLECTOR, uiValue := 2)
    Frame (0,60 80x30)
        shows SelSort(uiSel := uiSort, stSearch := stSearch, ITF_SPERRAT_COLLECTOR := ITF_SPERRAT_COLLECTOR, uiValue := 1)
END_VISUALIZATION

// 40 Visualizations/COLLECTOR/Help Funktionen/SortPfeil
VISUALIZATION SortPfeil  // 15x15
    Image (0,0 15x15), image: CtaVisSymbols.ImagePool.arrow-down_solo_black
END_VISUALIZATION

// 40 Visualizations/POPUP/SperrAntrieb_POPUP
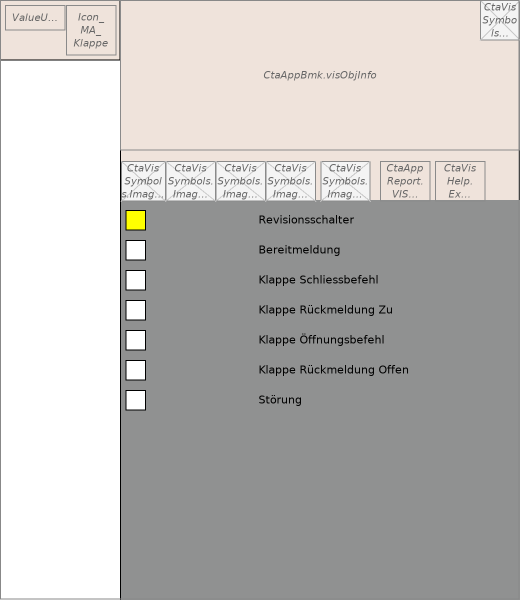
VISUALIZATION SperrAntrieb_POPUP  // 520x600
VAR_INPUT
    ITF_SPERRANTRIEBIN  :   ITF_SPERRANTRIEB;
    stExklParameter		:   STRING[40];	
	uiPopUpGruppe		: UINT;
END_VAR
    Rectangle (0,0 120x60)
    Rectangle (120,0 400x600)
    Frame (120,0 400x150)
        shows CtaAppBmk.visObjInfo(ITF_BMK_IN := ITF_SPERRANTRIEBIN)
    Image (480,0 40x40), image: CtaVisSymbols.ImagePool.close_solo_black
        OnMouseClick:  Dialog=SperrAntrieb_POPUP, Result=None, NumpadKeypadSet=True
    Frame (121,200 399x400), frame switch variable: uiPopUpGruppe
        shows SperrAntrieb_OVERVIEW(ITF_SPERRANTRIEBIN := ITF_SPERRANTRIEBIN)
        shows SperrAntrieb_MANUAL(ITF_SPERRANTRIEBIN := ITF_SPERRANTRIEBIN)
        shows SperrAntrieb_PARAMETER(ITF_SPERRANTRIEBIN := ITF_SPERRANTRIEBIN)
        shows SperrAntrieb_IO(ITF_SPERRANTRIEBIN := ITF_SPERRANTRIEBIN)
        shows SperrAntrieb_BUS(ITF_SPERRANTRIEBIN := ITF_SPERRANTRIEBIN)
        shows SperrAntrieb_REPORTS(ITF_SPERRANTRIEBIN := ITF_SPERRANTRIEBIN)
        pReferences[2]: ITF_Parameter=ITF_SPERRANTRIEBIN.proParameter
    Frame (121,161 399x40)
        shows SperrAntrieb_PopUpListe(uiPopUpGruppe := uiPopUpGruppe, xHand := ITF_SPERRANTRIEBIN.proIsHandOnOrOff, xHandOff := ITF_SPERRANTRIEBIN.proHandOff, ITF_REPORTMANAGER_IN := ITF_SPERRANTRIEBIN.proITF_REPORTMANAGER, stExklParameter := stExklParameter)
        pReferences[0]: AnzError=ITF_SPERRANTRIEBIN.proAnzError, AnzWarning=ITF_SPERRANTRIEBIN.proAnzWarning
    Frame (5,5 110x50), input disabled if: TRUE, frame switch variable: ITF_SPERRANTRIEBIN.proValveIcon
        shows SperrAntrieb_MA_Flap_Txt_L_Above(ITF_SPERRANTRIEB_IN := ITF_SPERRANTRIEBIN, stExklParameter := stExklParameter)
        shows SperrAntrieb_MB_Flap_Txt_L_Below(ITF_SPERRANTRIEB_IN := ITF_SPERRANTRIEBIN, stExklParameter := stExklParameter)
        shows SperrAntrieb_ML_Flap_Txt_L_Above(ITF_SPERRANTRIEB_IN := ITF_SPERRANTRIEBIN, stExklParameter := stExklParameter)
        shows SperrAntrieb_ML_Flap_Txt_L_Below(ITF_SPERRANTRIEB_IN := ITF_SPERRANTRIEBIN, stExklParameter := stExklParameter)
        shows SperrAntrieb_MA_Flap_Txt_R_Above(ITF_SPERRANTRIEB_IN := ITF_SPERRANTRIEBIN, stExklParameter := stExklParameter)
        shows SperrAntrieb_MB_Flap_Right_Txt_R_Below(ITF_SPERRANTRIEB_IN := ITF_SPERRANTRIEBIN, stExklParameter := stExklParameter)
        shows SperrAntrieb_MR_Flap_Txt_R_Above(ITF_SPERRANTRIEB_IN := ITF_SPERRANTRIEBIN, stExklParameter := stExklParameter)
        shows SperrAntrieb_MR_Flap_Txt_R_Below(ITF_SPERRANTRIEB_IN := ITF_SPERRANTRIEBIN, stExklParameter := stExklParameter)
        shows S_AT_ML_Valve_AB_Down_Txt_L_Above(ITF_STELLANTRIEB_IN := ITF_STELLANTRIEBIN)
        shows S_AT_ML_Valve_AB_Down_Txt_L_Below(ITF_STELLANTRIEB_IN := ITF_STELLANTRIEBIN)
        shows S_AT_ML_Valve_AB_Up_Txt_L_Above(ITF_STELLANTRIEB_IN := ITF_STELLANTRIEBIN)
        shows S_AT_ML_Valve_AB_Up_Txt_L_Below(ITF_STELLANTRIEB_IN := ITF_STELLANTRIEBIN)
        shows S_AT_ML_Valve_Flow_Txt_L_Above(ITF_STELLANTRIEB_IN := ITF_STELLANTRIEBIN)
        shows S_AT_ML_Valve_Flow_Txt_L_Below(ITF_STELLANTRIEB_IN := ITF_STELLANTRIEBIN)
        shows S_AT_ML_Valve_Mix_Txt_L_Above(ITF_STELLANTRIEB_IN := ITF_STELLANTRIEBIN)
        shows S_AT_ML_Valve_Mix_Txt_L_Below(ITF_STELLANTRIEB_IN := ITF_STELLANTRIEBIN)
        shows S_AT_MA_Valve_AB_Left_Txt_R_Above(ITF_STELLANTRIEB_IN := ITF_STELLANTRIEBIN)
        shows S_AT_MA_Valve_AB_Right_Txt_R_Above(ITF_STELLANTRIEB_IN := ITF_STELLANTRIEBIN)
        shows S_AT_MA_Valve_Flow_Txt_R_Above(ITF_STELLANTRIEB_IN := ITF_STELLANTRIEBIN)
        shows S_AT_MA_Valve_Mix_Txt_R_Above(ITF_STELLANTRIEB_IN := ITF_STELLANTRIEBIN)
        shows S_AT_MB_Valve_AB_Left_Txt_R_Below(ITF_STELLANTRIEB_IN := ITF_STELLANTRIEBIN)
        shows S_AT_MB_Valve_AB_Right_Txt_R_Below(ITF_STELLANTRIEB_IN := ITF_STELLANTRIEBIN)
        shows S_AT_MB_Valve_Flow_Txt_R_Below(ITF_STELLANTRIEB_IN := ITF_STELLANTRIEBIN)
        shows S_AT_MB_Valve_Mix_Txt_R_Below(ITF_STELLANTRIEB_IN := ITF_STELLANTRIEBIN)
        shows S_AT_MR_Valve_AB_Down_Txt_R_Above(ITF_STELLANTRIEB_IN := ITF_STELLANTRIEBIN)
        shows S_AT_MR_Valve_AB_Down_Txt_R_Below(ITF_STELLANTRIEB_IN := ITF_STELLANTRIEBIN)
        shows S_AT_MR_Valve_AB_Up_Txt_R_Above(ITF_STELLANTRIEB_IN := ITF_STELLANTRIEBIN)
        shows S_AT_MR_Valve_AB_Up_Txt_R_Below(ITF_STELLANTRIEB_IN := ITF_STELLANTRIEBIN)
        shows S_AT_MR_Valve_Flow_Txt_R_Above(ITF_STELLANTRIEB_IN := ITF_STELLANTRIEBIN)
        shows S_AT_MR_Valve_Flow_Txt_R_Below(ITF_STELLANTRIEB_IN := ITF_STELLANTRIEBIN)
        shows S_AT_MR_Valve_Mix_Txt_R_Above(ITF_STELLANTRIEB_IN := ITF_STELLANTRIEBIN)
        shows S_AT_MR_Valve_Mix_Txt_R_Below(ITF_STELLANTRIEB_IN := ITF_STELLANTRIEBIN)
        shows S_AT_MR_Valve_AB_Up_Txt_R_Above()
        shows S_AT_MR_Valve_AB_Up_Txt_R_Below()
        shows S_AT_MR_Flap_Txt_R_Above()
        shows S_AT_MR_Flap_Txt_R_Below()
        shows S_AT_MR_Valve_Flow_Txt_R_Above()
        shows S_AT_MR_Valve_Flow_Txt_R_Below()
        shows S_AT_MR_Valve_Mix_Txt_R_Above()
        shows S_AT_MR_Valve_Mix_Txt_R_Below()
END_VISUALIZATION

// 40 Visualizations/POPUP/SperrAntrieb_PopUpListe
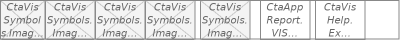
VISUALIZATION SperrAntrieb_PopUpListe  // 400x40
VAR_IN_OUT
	uiPopUpGruppe : UINT;
END_VAR
VAR_INPUT
    xHand           		: BOOL;
    xHandOff        		: BOOL;
    ITF_REPORTMANAGER_IN    : CtaAppReport.ITF_REPORTMANAGER;
    stExklParameter     	: STRING[40];
END_VAR
    Rectangle (100,0 40x40), colour toggle: uiPopUpGruppe = 2
        OnMouseDown: execute { uiPopUpGruppe := 2; }
    Rectangle (50,0 40x40), colour toggle: uiPopUpGruppe = 1
        OnMouseDown: execute { uiPopUpGruppe := 1; }
    Rectangle (0,0 40x40), colour toggle: uiPopUpGruppe = 0
        OnMouseDown: execute { uiPopUpGruppe := 0; }
    Image (0,0 45x40), image: CtaVisSymbols.ImagePool.eye
        OnMouseDown: execute { uiPopUpGruppe := 0; }
    Image (45,0 50x40), image: CtaVisSymbols.ImagePool.front_hand_Black
        OnMouseDown: execute { uiPopUpGruppe := 1; }
    Image (95,0 50x40), image: CtaVisSymbols.ImagePool.gear
        OnMouseDown: execute { uiPopUpGruppe := 2; }
    Image (45,0 50x40), invisible if: NOT xHand, image: CtaVisSymbols.ImagePool.front_hand_Yellow
        OnMouseDown: execute { uiPopUpGruppe := 1; }
    Rectangle (205,0 40x40), colour toggle: uiPopUpGruppe = 4
        OnMouseDown: execute { uiPopUpGruppe := 4; }
    Image (200,0 50x40), image: CtaVisSymbols.ImagePool.lan
        OnMouseDown: execute { uiPopUpGruppe := 4; }
    Image (45,0 50x40), invisible if: NOT xHandOff, image: CtaVisSymbols.ImagePool.front_hand_Yellow_Off
        OnMouseDown: execute { uiPopUpGruppe := 1; }
    Rectangle (150,0 40x40), colour toggle: uiPopUpGruppe = 3
        OnMouseDown: execute { uiPopUpGruppe := 3; }
    Image (145,0 50x40), image: CtaVisSymbols.ImagePool.dip-switch
        OnMouseDown: execute { uiPopUpGruppe := 3; }
    Rectangle (260,0 50x40), colour toggle: uiPopUpGruppe = 5
        OnMouseDown: execute { uiPopUpGruppe := 5; }
    Frame (260,0 50x40)
        shows CtaAppReport.VIS_ANZ_REPORTS_MODUL(ITF_REPORTMANAGER_IN := ITF_REPORTMANAGER_IN)
        OnMouseClick: execute { uiPopUpGruppe := 5; }
    Rectangle (315,0 50x40), colour toggle: uiPopUpGruppe = 6
        OnMouseDown: execute { uiPopUpGruppe := 6; }
    Frame (315,0 50x40)
        shows CtaVisHelp.ExkParameterSymbol(stExklParameter := stExklParameter)
END_VISUALIZATION

// 40 Visualizations/ICON/SperrAntrieb_BASE/Icons/Motor
VISUALIZATION Motor  // 15x15
VAR_INPUT
    ITF_SPERRANTRIEB_IN   :   ITF_SPERRANTRIEB;	
END_VAR
    Ellipse (0,0 15x15), "M", colour toggle: ITF_SPERRANTRIEB_IN.proIsError
    Ellipse (0,0 15x15), "M", colour toggle: ITF_SPERRANTRIEB_IN.proOn, invisible if: ITF_SPERRANTRIEB_IN.proIsError
END_VISUALIZATION

// 40 Visualizations/POPUP/PARAMETER/SperrAntrieb_PARAMETER
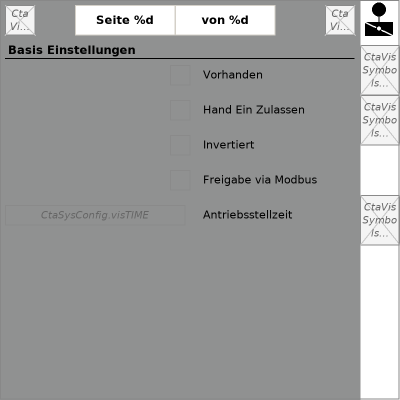
VISUALIZATION SperrAntrieb_PARAMETER  // 400x400
VAR_INPUT
    ITF_SPERRANTRIEBIN : ITF_SPERRANTRIEB;
END_VAR
VAR
    uiParameterGruppe : UINT;
END_VAR
    Image (145,122 150x30), image: ImagePool.Kreis
    Frame (360,0 40x300)
        shows SperrAntrieb_ParameterListe(uiParameterGruppe := uiParameterGruppe)
    Frame (0,0 360x400), frame switch variable: uiParameterGruppe
        shows SperrAntrieb_ParameterBase(ITF_SPERRANTRIEBIN := ITF_SPERRANTRIEBIN)
        shows SperrAntrieb_ParameterFuses(ITF_SPERRANTRIEBIN := ITF_SPERRANTRIEBIN)
        shows SperrAntrieb_ParameterIO(ITF_SPERRANTRIEBIN := ITF_SPERRANTRIEBIN)
        shows SperrAntrieb_ParameterInfluxDb(ITF_SPERRANTRIEBIN := ITF_SPERRANTRIEBIN)
        shows S_AT_ParameterInfluxDb(ITF_Parameter := ITF_Parameter)
        pReferences[0]: ITF_Parameter=ITF_Parameter
        pReferences[1]: ITF_Parameter=ITF_Parameter
        pReferences[2]: ITF_Parameter=ITF_Parameter
        pReferences[3]: ITF_Parameter=ITF_Parameter
END_VISUALIZATION

// 40 Visualizations/POPUP/PARAMETER/SperrAntrieb_ParameterListe
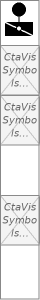
VISUALIZATION SperrAntrieb_ParameterListe  // 40x300
VAR_IN_OUT
	uiParameterGruppe : UINT;
END_VAR
    Rectangle (0,100 39x40), colour toggle: uiParameterGruppe = 2
        OnMouseDown: execute { uiParameterGruppe := 2; }
    Rectangle (0,50 39x40), colour toggle: uiParameterGruppe = 1
        OnMouseDown: execute { uiParameterGruppe := 1; }
    Rectangle (0,0 39x40), colour toggle: uiParameterGruppe = 0
        OnMouseDown: execute { uiParameterGruppe := 0; }
    Image (0,45 40x50), image: CtaVisSymbols.ImagePool.lightning-bolt-circle
        OnMouseDown: execute { uiParameterGruppe := 1; }
    Image (0,95 40x50), image: CtaVisSymbols.ImagePool.dip-switch
        OnMouseDown: execute { uiParameterGruppe := 2; }
    Rectangle (0,200 39x40), colour toggle: uiParameterGruppe = 3
        OnMouseDown: execute { uiParameterGruppe := 3; }
    Image (0,195 40x50), image: CtaVisSymbols.ImagePool.sine-wave
        OnMouseDown: execute { uiParameterGruppe := 3; }
    Frame (0,0 39x40)
        shows SperrAntrieb_Icon_SperrAntrieb()
        OnMouseDown: execute { uiParameterGruppe := 0; }
END_VISUALIZATION

// 40 Visualizations/POPUP/MANUAL/SperrAntrieb_MANUAL
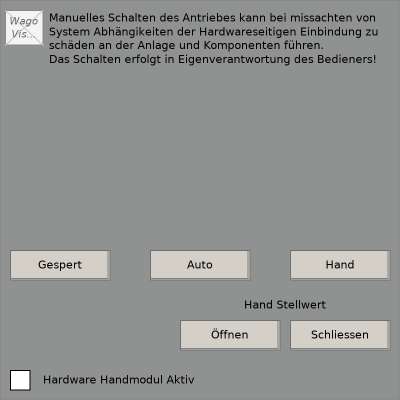
VISUALIZATION SperrAntrieb_MANUAL  // 400x400
VAR_INPUT
    ITF_SPERRANTRIEBIN    :   ITF_SPERRANTRIEB;	
END_VAR
    Button (10,250 100x30), "Gespert", colour toggle: ITF_SPERRANTRIEBIN.proHandOff, pressed state: ITF_SPERRANTRIEBIN.proHandOff
        toggle ITF_SPERRANTRIEBIN.proHandOff
    Button (290,250 100x30), "Hand", colour toggle: ITF_SPERRANTRIEBIN.proHandOn, pressed state: ITF_SPERRANTRIEBIN.proHandOn
        toggle ITF_SPERRANTRIEBIN.proHandOn
    Button (150,250 100x30), "Auto", colour toggle: ITF_SPERRANTRIEBIN.proAuto, pressed state: ITF_SPERRANTRIEBIN.proAuto
        toggle ITF_SPERRANTRIEBIN.proAuto
    Label (46,10 350x100), "Manuelles Schalten des Antriebes kann bei missachten von System Abhängikeiten der Hardwareseitigen Einbindung zu schäden an der Anlage und Komponenten führen. Das Schalten erfolgt in Eigenverantwortung des Bedieners!"
    Image (5,10 38x35), image: WagoVisuIcons.WagoIcons.2
    Label (235,295 100x20), "Hand Stellwert"
    Rectangle (10,370 20x20), colour toggle: ITF_SPERRANTRIEBIN.proHardWareHandModulAktive, invisible if: NOT ITF_SPERRANTRIEBIN.proHardWareHandModulAktive
    Label (40,370 200x20), "Hardware Handmodul Aktiv", invisible if: NOT ITF_SPERRANTRIEBIN.proHardWareHandModulAktive
    Button (290,320 100x30), "Schliessen", colour toggle: ITF_SPERRANTRIEBIN.proHandManualClose, pressed state: ITF_SPERRANTRIEBIN.proHandManualClose, invisible if: NOT ITF_SPERRANTRIEBIN.proHandOn
        toggle ITF_SPERRANTRIEBIN.proHandManualClose
    Button (180,320 100x30), "Öffnen", colour toggle: ITF_SPERRANTRIEBIN.proHandManualOpen, pressed state: ITF_SPERRANTRIEBIN.proHandManualOpen, invisible if: NOT ITF_SPERRANTRIEBIN.proHandOn
        toggle ITF_SPERRANTRIEBIN.proHandManualOpen
END_VISUALIZATION

// 40 Visualizations/POPUP/OVERVIEW/SperrAntrieb_OVERVIEW
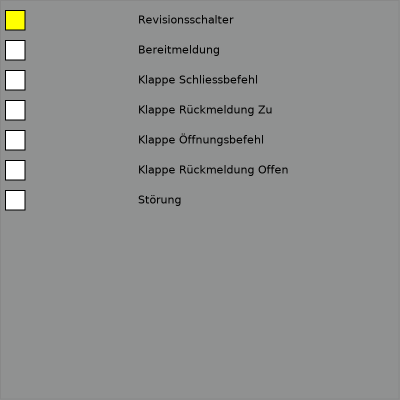
VISUALIZATION SperrAntrieb_OVERVIEW  // 400x400
VAR_INPUT
    ITF_SPERRANTRIEBIN    :   ITF_SPERRANTRIEB;	
END_VAR
    Label (135,10 200x20), "Revisionsschalter"
    Label (135,40 200x20), "Bereitmeldung"
    Rectangle (5,10 20x20), colour toggle: ITF_SPERRANTRIEBIN.proRevisionSwitchOk
    Rectangle (5,40 20x20), colour toggle: ITF_SPERRANTRIEBIN.proIsReady
    Rectangle (5,70 20x20), colour toggle: ITF_SPERRANTRIEBIN.proOnZu
    Label (135,70 200x20), "Klappe Schliessbefehl"
    Rectangle (5,100 20x20), colour toggle: ITF_SPERRANTRIEBIN.proRükIsClosed, invisible if: ITF_SPERRANTRIEBIN.proNotShowDI_RükIsClosed
    Label (135,100 200x20), "Klappe Rückmeldung Zu", invisible if: ITF_SPERRANTRIEBIN.proNotShowDI_RükIsClosed
    Rectangle (5,130 20x20), colour toggle: ITF_SPERRANTRIEBIN.proOnAuf
    Label (135,130 200x20), "Klappe Öffnungsbefehl"
    Rectangle (5,160 20x20), colour toggle: ITF_SPERRANTRIEBIN.proRükIsOpen, invisible if: ITF_SPERRANTRIEBIN.proNotShowDI_RükIsOpen
    Label (135,160 200x20), "Klappe Rückmeldung Offen", invisible if: ITF_SPERRANTRIEBIN.proNotShowDI_RükIsOpen
    Rectangle (5,190 20x20), colour toggle: ITF_SPERRANTRIEBIN.proIsError
    Label (135,190 200x20), "Störung"
END_VISUALIZATION

// 40 Visualizations/POPUP/BUS/SperrAntrieb_BUS
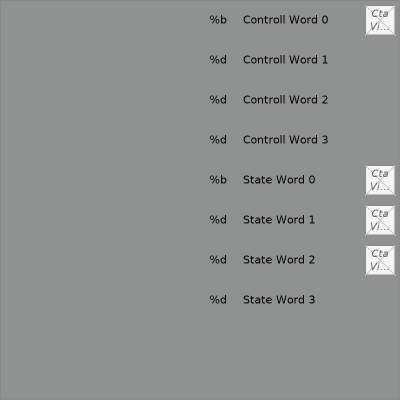
VISUALIZATION SperrAntrieb_BUS  // 400x400
VAR_INPUT
    ITF_SPERRANTRIEBIN    :   ITF_SPERRANTRIEB;	
END_VAR
    Frame (100,0 300x350)
        shows SperrAntrieb_BUS_CS(ITF_SPERRANTRIEBIn := ITF_SPERRANTRIEBIN, ayControllWord := ITF_SPERRANTRIEBIN.proModbusControllWord, ayStateWord := ITF_SPERRANTRIEBIN.proModbusStateWord)
END_VISUALIZATION

// 40 Visualizations/POPUP/BUS/SperrAntrieb_BUS_SW0_Detail
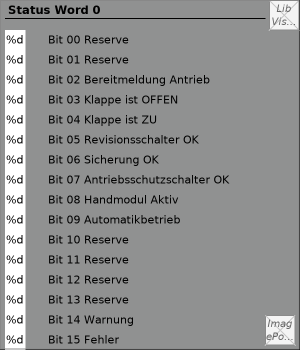
VISUALIZATION SperrAntrieb_BUS_SW0_Detail  // 300x350
VAR_IN_OUT
    wDetail     :   WORD;
END_VAR
VAR_INPUT	
    ITF_SPERRANTRIEBIN    :   ITF_SPERRANTRIEB;
END_VAR
VAR_IN_OUT
    xShow       :   BOOL;
END_VAR
    Rectangle (0,0 300x350)
    Textfield (5,30 20x20), "%d", text variable: TO_WORD(wDetail.0), input disabled if: NOT ITF_SPERRANTRIEBIn.proModbusTest
        OnMouseClick: execute { wDetail.0 := NOT wDetail.0; }
    Label (45,30 180x20), "Bit 00 Reserve"
    Textfield (5,50 20x20), "%d", text variable: TO_WORD(wDetail.1), input disabled if: NOT ITF_SPERRANTRIEBIn.proModbusTest
        OnMouseClick: execute { wDetail.1 := NOT wDetail.1; }
    Label (45,50 180x20), "Bit 01 Reserve"
    Textfield (5,70 20x20), "%d", text variable: TO_WORD(wDetail.2), input disabled if: NOT ITF_SPERRANTRIEBIn.proModbusTest
        OnMouseClick: execute { wDetail.2 := NOT wDetail.2; }
    Label (45,70 180x20), "Bit 02 Bereitmeldung Antrieb"
    Textfield (5,90 20x20), "%d", text variable: TO_WORD(wDetail.3), input disabled if: NOT ITF_SPERRANTRIEBIn.proModbusTest
        OnMouseClick: execute { wDetail.3 := NOT wDetail.3; }
    Label (45,90 180x20), "Bit 03 Klappe ist OFFEN"
    Textfield (5,110 20x20), "%d", text variable: TO_WORD(wDetail.4), input disabled if: NOT ITF_SPERRANTRIEBIn.proModbusTest
        OnMouseClick: execute { wDetail.4 := NOT wDetail.4; }
    Label (45,110 180x20), "Bit 04 Klappe ist ZU"
    Textfield (5,130 20x20), "%d", text variable: TO_WORD(wDetail.5), input disabled if: NOT ITF_SPERRANTRIEBIn.proModbusTest
        OnMouseClick: execute { wDetail.5 := NOT wDetail.5; }
    Label (45,130 180x20), "Bit 05 Revisionsschalter OK"
    Textfield (5,150 20x20), "%d", text variable: TO_WORD(wDetail.6), input disabled if: NOT ITF_SPERRANTRIEBIn.proModbusTest
        OnMouseClick: execute { wDetail.6 := NOT wDetail.6; }
    Label (45,150 180x20), "Bit 06 Sicherung OK"
    Textfield (5,170 20x20), "%d", text variable: TO_WORD(wDetail.7), input disabled if: NOT ITF_SPERRANTRIEBIn.proModbusTest
        OnMouseClick: execute { wDetail.7 := NOT wDetail.7; }
    Label (45,170 180x20), "Bit 07 Antriebsschutzschalter OK"
    Textfield (5,190 20x20), "%d", text variable: TO_WORD(wDetail.8), input disabled if: NOT ITF_SPERRANTRIEBIn.proModbusTest
        OnMouseClick: execute { wDetail.8 := NOT wDetail.8; }
    Label (45,190 180x20), "Bit 08 Handmodul Aktiv"
    Textfield (5,210 20x20), "%d", text variable: TO_WORD(wDetail.9), input disabled if: NOT ITF_SPERRANTRIEBIn.proModbusTest
        OnMouseClick: execute { wDetail.9 := NOT wDetail.9; }
    Label (45,210 180x20), "Bit 09 Automatikbetrieb"
    Textfield (5,230 20x20), "%d", text variable: TO_WORD(wDetail.10), input disabled if: NOT ITF_SPERRANTRIEBIn.proModbusTest
        OnMouseClick: execute { wDetail.10 := NOT wDetail.10; }
    Label (45,230 180x20), "Bit 10 Reserve"
    Textfield (5,250 20x20), "%d", text variable: TO_WORD(wDetail.11), input disabled if: NOT ITF_SPERRANTRIEBIn.proModbusTest
        OnMouseClick: execute { wDetail.11 := NOT wDetail.11; }
    Label (45,250 180x20), "Bit 11 Reserve"
    Textfield (5,270 20x20), "%d", text variable: TO_WORD(wDetail.12), input disabled if: NOT ITF_SPERRANTRIEBIn.proModbusTest
        OnMouseClick: execute { wDetail.12 := NOT wDetail.12; }
    Label (45,270 180x20), "Bit 12 Reserve"
    Textfield (5,290 20x20), "%d", text variable: TO_WORD(wDetail.13), input disabled if: NOT ITF_SPERRANTRIEBIn.proModbusTest
        OnMouseClick: execute { wDetail.13 := NOT wDetail.13; }
    Label (45,290 180x20), "Bit 13 Reserve"
    Textfield (5,310 20x20), "%d", text variable: TO_WORD(wDetail.14), input disabled if: NOT ITF_SPERRANTRIEBIn.proModbusTest
        OnMouseClick: execute { wDetail.14 := NOT wDetail.14; }
    Label (45,310 180x20), "Bit 14 Warnung"
    Textfield (5,330 20x20), "%d", text variable: TO_WORD(wDetail.15), input disabled if: NOT ITF_SPERRANTRIEBIn.proModbusTest
        OnMouseClick: execute { wDetail.15 := NOT wDetail.15; }
    Label (45,330 180x20), "Bit 15 Fehler"
    Image (269,0 30x30), image: LibVis01VisuBasic.imgpVisuCTA.close_solo_black
        OnMouseClick: execute { xShow := FALSE; ITF_SPERRANTRIEBIN.proModbusTest := FALSE; }
    Label (5,0 150x20), "Status Word 0"
    Image (265,315 30x30), invisible if: ITF_SPERRANTRIEBIN.proModbusTest, image: ImagePool.front_hand_FILL0_wght400_GRAD0_opsz48
        OnMouseClick: execute { ITF_SPERRANTRIEBIN.proModbusTest := TRUE; }
    Image (265,315 30x30), invisible if: NOT ITF_SPERRANTRIEBIN.proModbusTest, image: ImagePool.front_hand_FILL0_wght400_GRAD0_opsz48Yellow
        OnMouseClick: execute { ITF_SPERRANTRIEBIN.proModbusTest := False; }
    Line (5,18) (265,18)
END_VISUALIZATION

// 40 Visualizations/POPUP/BUS/SperrAntrieb_BUS_CW0_Detail
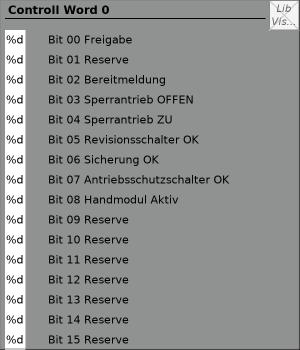
VISUALIZATION SperrAntrieb_BUS_CW0_Detail  // 300x350
VAR_IN_OUT
    wDetail :   WORD;
END_VAR
VAR_IN_OUT
    xShow   :   BOOL;
END_VAR
    Rectangle (0,0 300x350)
    Textfield (5,30 20x20), "%d", text variable: TO_WORD(wDetail.0), input disabled if: TRUE
    Label (45,30 180x20), "Bit 00 Freigabe"
    Textfield (5,50 20x20), "%d", text variable: TO_WORD(wDetail.1), input disabled if: TRUE
    Label (45,50 180x20), "Bit 01 Reserve"
    Textfield (5,70 20x20), "%d", text variable: TO_WORD(wDetail.2), input disabled if: TRUE
    Label (45,70 180x20), "Bit 02 Bereitmeldung"
    Textfield (5,90 20x20), "%d", text variable: TO_WORD(wDetail.3), input disabled if: TRUE
    Label (45,90 180x20), "Bit 03 Sperrantrieb OFFEN"
    Textfield (5,110 20x20), "%d", text variable: TO_WORD(wDetail.4), input disabled if: TRUE
    Label (45,110 180x20), "Bit 04 Sperrantrieb ZU"
    Textfield (5,130 20x20), "%d", text variable: TO_WORD(wDetail.5), input disabled if: TRUE
    Label (45,130 180x20), "Bit 05 Revisionsschalter OK"
    Textfield (5,150 20x20), "%d", text variable: TO_WORD(wDetail.6), input disabled if: TRUE
    Label (45,150 180x20), "Bit 06 Sicherung OK"
    Textfield (5,170 20x20), "%d", text variable: TO_WORD(wDetail.7), input disabled if: TRUE
    Label (45,170 180x20), "Bit 07 Antriebsschutzschalter OK"
    Textfield (5,190 20x20), "%d", text variable: TO_WORD(wDetail.8), input disabled if: TRUE
    Label (45,190 180x20), "Bit 08 Handmodul Aktiv"
    Textfield (5,210 20x20), "%d", text variable: TO_WORD(wDetail.9), input disabled if: TRUE
    Label (45,210 180x20), "Bit 09 Reserve"
    Textfield (5,230 20x20), "%d", text variable: TO_WORD(wDetail.10), input disabled if: TRUE
    Label (45,230 180x20), "Bit 10 Reserve"
    Textfield (5,250 20x20), "%d", text variable: TO_WORD(wDetail.11), input disabled if: TRUE
    Label (45,250 180x20), "Bit 11 Reserve"
    Textfield (5,270 20x20), "%d", text variable: TO_WORD(wDetail.12), input disabled if: TRUE
    Label (45,270 180x20), "Bit 12 Reserve"
    Textfield (5,290 20x20), "%d", text variable: TO_WORD(wDetail.13), input disabled if: TRUE
    Label (45,290 180x20), "Bit 13 Reserve"
    Textfield (5,310 20x20), "%d", text variable: TO_WORD(wDetail.14), input disabled if: TRUE
    Label (45,310 180x20), "Bit 14 Reserve"
    Textfield (5,330 20x20), "%d", text variable: TO_WORD(wDetail.15), input disabled if: TRUE
    Label (45,330 180x20), "Bit 15 Reserve"
    Image (269,0 30x30), image: LibVis01VisuBasic.imgpVisuCTA.close_solo_black
        OnMouseClick: execute { xShow := FALSE; }
    Label (5,0 150x20), "Controll Word 0"
    Line (5,18) (265,18)
END_VISUALIZATION

// 40 Visualizations/POPUP/BUS/SperrAntrieb_BUS_CS
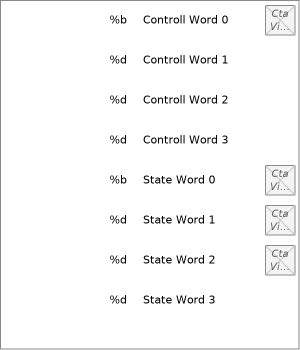
VISUALIZATION SperrAntrieb_BUS_CS  // 300x350
VAR_INPUT
    ITF_SPERRANTRIEBIn        :   ITF_SPERRANTRIEB;
    ayControllWord  :   REFERENCE TO ARRAY[0..3] OF WORD;
    ayStateWord     :   REFERENCE TO ARRAY[0..3] OF WORD;
END_VAR
VAR
    xShowCw :   BOOL;
    xShowSw :   BOOL;
    xShowSw1:   BOOL;
    xShowSw2:   BOOL;
END_VAR
    Textfield (0,10 130x20), "%b", text variable: ayControllWord[0]
    Label (140,10 120x20), "Controll Word 0"
    Label (140,50 120x20), "Controll Word 1"
    Textfield (0,50 130x20), "%d", text variable: ayControllWord[1]
    Label (140,90 120x20), "Controll Word 2", invisible if: TRUE
    Textfield (0,90 130x20), "%d", text variable: ayControllWord[2], invisible if: TRUE
    Label (140,130 120x20), "Controll Word 3", invisible if: TRUE
    Textfield (0,130 130x20), "%d", text variable: ayControllWord[3], invisible if: TRUE
    Image (265,5 30x30), image: CtaVisSymbols.ImagePool.information-variant
        OnMouseClick: execute {
            xShowCw := TRUE;
            xShowSw := FALSE;
            xShowSw1:= FALSE;
            xShowSw2:= FALSE;
        }
    Frame (300,0 300x350), invisible if: NOT xShowCw
        shows SperrAntrieb_BUS_CW0_Detail(wDetail := ayControllWord[0], xShow := xShowCw)
    Label (140,290 120x20), "State Word 3", invisible if: TRUE
    Textfield (0,170 130x20), "%b", text variable: ayStateWord[0]
        OnMouseDown: write the text variable via Default
    Label (140,170 120x20), "State Word 0"
    Label (140,210 120x20), "State Word 1"
    Textfield (0,210 130x20), "%d", text variable: ayStateWord[1]
    Label (140,250 120x20), "State Word 2"
    Textfield (0,250 130x20), "%d", text variable: ayStateWord[2]
    Textfield (0,290 130x20), "%d", text variable: ayStateWord[3], invisible if: TRUE
    Image (265,165 30x30), image: CtaVisSymbols.ImagePool.information-variant
        OnMouseClick: execute {
            xShowCw := FALSE;
            xShowSw := TRUE;
            xShowSw1:= FALSE;
            xShowSw2:= FALSE;
        }
    Frame (300,0 300x350), invisible if: NOT xShowSw
        shows SperrAntrieb_BUS_SW0_Detail(wDetail := ayStateWord[0], ITF_SPERRANTRIEBIN := ITF_SPERRANTRIEBIn, xShow := xShowSw2)
    Image (265,205 30x30), image: CtaVisSymbols.ImagePool.information-variant
        OnMouseClick: execute {
            xShowCw := FALSE;
            xShowSw := FALSE;
            xShowSw1:= TRUE;
            xShowSw2:= FALSE;
        }
    Frame (300,0 300x350), invisible if: NOT xShowSw1
        shows SperrAntrieb_BUS_SW1_Detail(wDetail := ayStateWord[1], ITF_SPERRANTRIEBIN := ITF_SPERRANTRIEBIn, xShow := xShowSw1)
    Frame (300,0 300x350), invisible if: NOT xShowSw2
        shows SperrAntrieb_BUS_SW2_Detail(wDetail := ayStateWord[2], ITF_SPERRANTRIEBIN := ITF_SPERRANTRIEBIn, xShow := xShowSw2)
        shows SperrAntrieb_BUS_SW2_Detail()
    Image (265,245 30x30), image: CtaVisSymbols.ImagePool.information-variant
        OnMouseClick: execute {
            xShowCw := FALSE;
            xShowSw := FALSE;
            xShowSw1:= FALSE;
            xShowSw2:= TRUE;
        }
END_VISUALIZATION

// 40 Visualizations/POPUP/BUS/SperrAntrieb_BUS_SW1_Detail
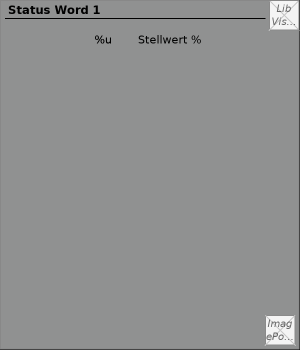
VISUALIZATION SperrAntrieb_BUS_SW1_Detail  // 300x350
VAR_IN_OUT
    wDetail     :   WORD;
END_VAR
VAR_INPUT	
    ITF_SPERRANTRIEBIN    :   ITF_SPERRANTRIEB;
END_VAR
VAR_IN_OUT
    xShow       :   BOOL;
END_VAR
    Rectangle (0,0 300x350)
    Image (269,0 30x30), image: LibVis01VisuBasic.imgpVisuCTA.close_solo_black
        OnMouseClick: execute { xShow := FALSE; ITF_SPERRANTRIEBIN.proModbusTest := FALSE; }
    Label (5,0 150x20), "Status Word 1"
    Image (265,315 30x30), invisible if: ITF_SPERRANTRIEBIN.proModbusTest, image: ImagePool.front_hand_FILL0_wght400_GRAD0_opsz48
        OnMouseClick: execute { ITF_SPERRANTRIEBIN.proModbusTest := TRUE; }
    Image (265,315 30x30), invisible if: NOT ITF_SPERRANTRIEBIn.proModbusTest, image: ImagePool.front_hand_FILL0_wght400_GRAD0_opsz48Yellow
        OnMouseClick: execute { ITF_SPERRANTRIEBIN.proModbusTest := False; }
    Label (135,30 120x20), "Stellwert %"
    Textfield (5,30 110x20), "%u", text variable: wDetail, input disabled if: NOT ITF_SPERRANTRIEBIn.proModbusTest
        OnMouseClick: write the text variable via InputWithLimits, min 0, max 100
    Textfield (5,30 110x20), "%u", text variable: wDetail, invisible if: ITF_SPERRANTRIEBIN.proModbusTest
    Line (5,18) (265,18)
END_VISUALIZATION

// 40 Visualizations/POPUP/BUS/SperrAntrieb_BUS_SW2_Detail
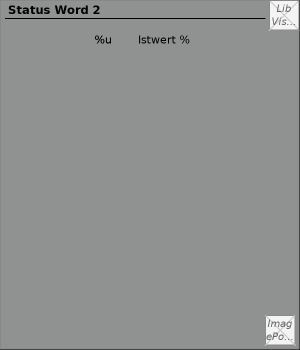
VISUALIZATION SperrAntrieb_BUS_SW2_Detail  // 300x350
VAR_IN_OUT
    wDetail             :   WORD;
END_VAR
VAR_INPUT	
    ITF_SPERRANTRIEBIN       :   ITF_SPERRANTRIEB;
END_VAR
VAR_IN_OUT
    xShow               :   BOOL;
END_VAR
    Rectangle (0,0 300x350)
    Image (269,0 30x30), image: LibVis01VisuBasic.imgpVisuCTA.close_solo_black
        OnMouseClick: execute { xShow := FALSE; ITF_SPERRANTRIEBIN.proModbusTest := FALSE; }
    Label (5,0 150x20), "Status Word 2"
    Image (265,315 30x30), invisible if: ITF_SPERRANTRIEBIn.proModbusTest, image: ImagePool.front_hand_FILL0_wght400_GRAD0_opsz48
        OnMouseClick: execute { ITF_SPERRANTRIEBIN.proModbusTest := TRUE; }
    Image (265,315 30x30), invisible if: NOT ITF_SPERRANTRIEBIN.proModbusTest, image: ImagePool.front_hand_FILL0_wght400_GRAD0_opsz48Yellow
        OnMouseClick: execute { ITF_SPERRANTRIEBIN.proModbusTest := False; }
    Label (135,30 120x20), "Istwert %"
    Textfield (5,30 110x20), "%u", text variable: wDetail, input disabled if: NOT ITF_SPERRANTRIEBIn.proModbusTest
        OnMouseClick: write the text variable via InputWithLimits, min 0, max 100
    Textfield (5,30 110x20), "%u", text variable: wDetail, invisible if: ITF_SPERRANTRIEBIN.proModbusTest
    Line (5,18) (265,18)
END_VISUALIZATION

// 40 Visualizations/POPUP/REPORTS/SperrAntrieb_REPORTS
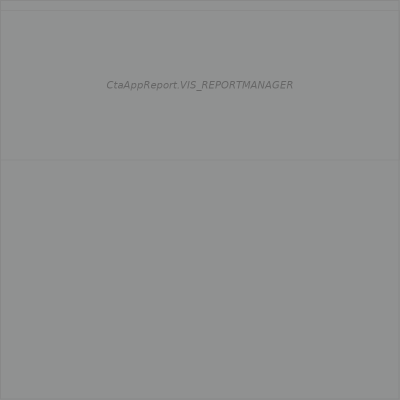
VISUALIZATION SperrAntrieb_REPORTS  // 400x400
VAR_INPUT
    ITF_SPERRANTRIEBIN    :   ITF_SPERRANTRIEB;	
END_VAR
    Frame (0,10 400x150)
        shows CtaAppReport.VIS_REPORTMANAGER(ITF_REPORTMANAGER := ITF_SPERRANTRIEBIN.proITF_REPORTMANAGER)
END_VISUALIZATION

// 40 Visualizations/POPUP/PARAMETER/SperrAntrieb_ParameterBase/SperrAntrieb_ParameterBase0
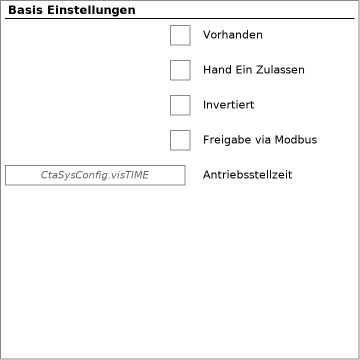
VISUALIZATION SperrAntrieb_ParameterBase0  // 360x360
VAR_INPUT
    ITF_SPERRANTRIEBIN : ITF_SPERRANTRIEB;
END_VAR
    Label (5,0 350x20), "Basis Einstellungen"
    Frame (170,25 20x20)
        shows CtaSysConfig.visBOOL(visfbBOOLIn := ITF_SPERRANTRIEBIN.p_scBase_fbxEnable)
    Label (200,25 150x20), "Vorhanden"
    Label (200,130 150x20), "Freigabe via Modbus"
    Frame (170,130 20x20)
        shows CtaSysConfig.visBOOL(visfbBOOLIn := ITF_SPERRANTRIEBIN.p_scBase_fbxControllMb)
    Frame (170,60 20x20)
        shows CtaSysConfig.visBOOL(visfbBOOLIn := ITF_SPERRANTRIEBIN.p_scManual_fbxAlowManualOn)
    Label (200,60 150x20), "Hand Ein Zulassen"
    Frame (170,95 20x20)
        shows CtaSysConfig.visBOOL(visfbBOOLIn := ITF_SPERRANTRIEBIN.p_scBase_fbxInvertiert)
    Label (200,95 150x20), "Invertiert"
    Label (200,165 150x20), "Antriebsstellzeit"
    Frame (5,165 180x20)
        shows CtaSysConfig.visTIME(visfbTIMEIn := ITF_SPERRANTRIEBIN.p_scBase_fbtSettingTime)
    Line (5,18) (354,18)
END_VISUALIZATION

// 40 Visualizations/POPUP/PARAMETER/SperrAntrieb_ParameterBase/SperrAntrieb_ParameterBase
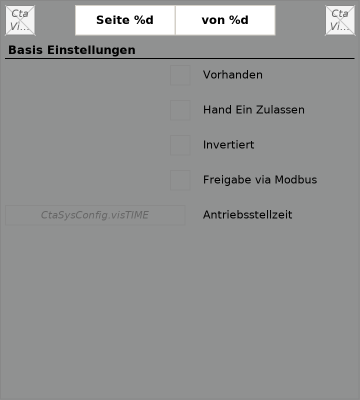
VISUALIZATION SperrAntrieb_ParameterBase  // 360x400
VAR_INPUT
    ITF_SPERRANTRIEBIN : ITF_SPERRANTRIEB;
END_VAR
VAR
    uiPage  :   UINT;
    uiMin   :   UINT    := 0;
    uiMax   :   UINT    := 0;
END_VAR
    Image (5,5 30x30), invisible if: uiPage = uiMin, image: CtaVisSymbols.ImagePool.arrow-left_square
        OnMouseClick: execute {
            uiPage := uiPage - 1;
            IF uiPage <= uiMin THEN
                uiPage := uiMin;
            END_IF;
        }
    Image (325,5 30x30), invisible if: uiPage = uiMax, image: CtaVisSymbols.ImagePool.arrow-right_square
        OnMouseClick: execute {
            uiPage := uiPage + 1;
            IF uiPage >= uiMax THEN
                uiPage := uiMax;
            END_IF;
        }
    Frame (0,40 360x360), frame switch variable: uiPage
        shows SperrAntrieb_ParameterBase0(ITF_SPERRANTRIEBIN := ITF_SPERRANTRIEBIN)
        shows S_AT_ParameterBase1()
        shows S_AT_ParameterBase3()
        shows SperrAT_ParameterBase1(ITF_Parameter := ITF_Parameter)
        pReferences[0]: ITF_Parameter=ITF_Parameter
        p982447995: ITF_Parameter
        p2498127594: ITF_Parameter
    Textfield (175,5 100x30), "von %d", text variable: uiMax
    Textfield (75,5 100x30), "Seite %d", text variable: uiPage
END_VISUALIZATION

// 40 Visualizations/POPUP/PARAMETER/SperrAntrieb_Fuse/SperrAntrieb_ParameterFuses0
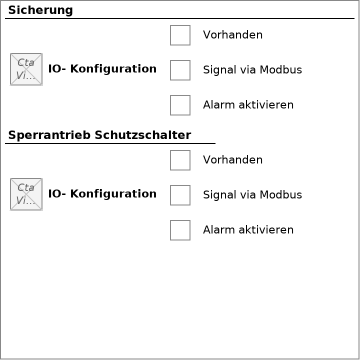
VISUALIZATION SperrAntrieb_ParameterFuses0  // 360x360
VAR_INPUT
    ITF_SPERRANTRIEBIN 	:	ITF_SPERRANTRIEB;
	ITF_Fuse_IN 		:	CtaSysIO.ITF_IO;
	ITF_ActuatorFuse_IN :	CtaSysIO.ITF_IO;
END_VAR
    Frame (170,25 20x20)
        shows CtaSysConfig.visBOOL(visfbBOOLIn := ITF_SPERRANTRIEBIN.p_scFuse_fbxEnable)
    Label (200,25 150x20), "Vorhanden"
    Frame (170,60 20x20)
        shows CtaSysConfig.visBOOL(visfbBOOLIn := ITF_SPERRANTRIEBIN.p_scFuse_fbxInputMb)
    Label (200,60 150x20), "Signal via Modbus"
    Frame (170,95 20x20)
        shows CtaSysConfig.visBOOL(visfbBOOLIn := ITF_SPERRANTRIEBIN.p_scFuse_fbxDoesAlarm)
    Label (200,95 150x20), "Alarm aktivieren"
    Label (5,0 350x20), "Sicherung"
    Label (5,125 350x20), "Sperrantrieb Schutzschalter"
    Frame (170,150 20x20)
        shows CtaSysConfig.visBOOL(visfbBOOLIn := ITF_SPERRANTRIEBIN.p_scActuatorFuse_fbxEnable)
    Label (200,150 150x20), "Vorhanden"
    Frame (170,185 20x20)
        shows CtaSysConfig.visBOOL(visfbBOOLIn := ITF_SPERRANTRIEBIN.p_scActuatorFuse_fbxInputMb)
    Label (200,185 150x20), "Signal via Modbus"
    Frame (170,220 20x20)
        shows CtaSysConfig.visBOOL(visfbBOOLIn := ITF_SPERRANTRIEBIN.p_scActuatorFuse_fbxDoesAlarm)
    Label (200,220 150x20), "Alarm aktivieren"
    Line (5,143) (215,143)
    Line (5,18) (354,18)
    Image (10,53 32x32), invisible if: ITF_Fuse_IN = 0, image: CtaVisSymbols.ImagePool.build
        OnMouseDown:  Dialog=SperrAntrieb_POPUP_IO_ITF, Parameters={ITF_IO_IN: ITF_Fuse_IN}, OpenModal=True, OpenCentered=True
    Label (45,59 120x20), "IO- Konfiguration", invisible if: ITF_Fuse_IN = 0
    Image (10,178 32x32), invisible if: ITF_ActuatorFuse_IN = 0, image: CtaVisSymbols.ImagePool.build
        OnMouseDown:  Dialog=SperrAntrieb_POPUP_IO_ITF, Parameters={ITF_IO_IN: ITF_ActuatorFuse_IN}, OpenModal=True, OpenCentered=True
    Label (45,184 120x20), "IO- Konfiguration", invisible if: ITF_ActuatorFuse_IN = 0
END_VISUALIZATION

// 40 Visualizations/POPUP/PARAMETER/SperrAntrieb_Fuse/SperrAntrieb_ParameterFuses
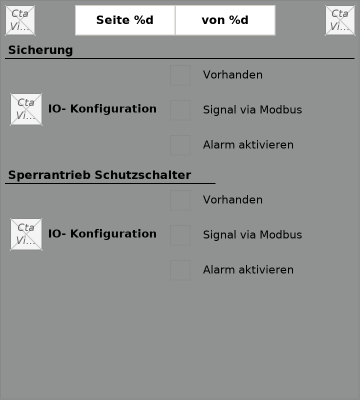
VISUALIZATION SperrAntrieb_ParameterFuses  // 360x400
VAR_INPUT
    ITF_SPERRANTRIEBIN : ITF_SPERRANTRIEB;
END_VAR
VAR
    uiPage  :   UINT;
    uiMin   :   UINT    := 0;
    uiMax   :   UINT    := 0;
END_VAR
    Image (5,5 30x30), invisible if: uiPage = uiMin, image: CtaVisSymbols.ImagePool.arrow-left_square
        OnMouseClick: execute {
            uiPage := uiPage - 1;
            IF uiPage <= uiMin THEN
                uiPage := uiMin;
            END_IF;
        }
    Image (325,5 30x30), invisible if: uiPage = uiMax, image: CtaVisSymbols.ImagePool.arrow-right_square
        OnMouseClick: execute {
            uiPage := uiPage + 1;
            IF uiPage >= uiMax THEN
                uiPage := uiMax;
            END_IF;
        }
    Frame (0,40 360x360), frame switch variable: uiPage
        shows SperrAntrieb_ParameterFuses0(ITF_SPERRANTRIEBIN := ITF_SPERRANTRIEBIN, ITF_Fuse_IN := ITF_SPERRANTRIEBIN.proFuse_ITF, ITF_ActuatorFuse_IN := ITF_SPERRANTRIEBIN.proActuatorFuse_ITF)
        shows AT_ParameterIO1(ITF_Parameter := ITF_Parameter)
        pReferences[0]: ITF_Parameter=ITF_Parameter
    Textfield (75,5 100x30), "Seite %d", text variable: uiPage
    Textfield (175,5 100x30), "von %d", text variable: uiMax
END_VISUALIZATION

// 40 Visualizations/POPUP/PARAMETER/SperrAntrieb_IO/SperrAntrieb_ParameterIO0
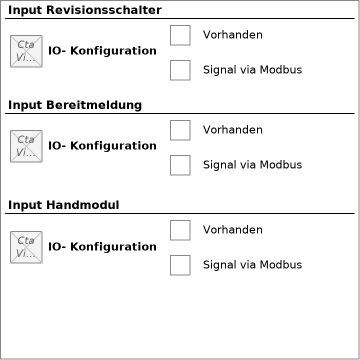
VISUALIZATION SperrAntrieb_ParameterIO0  // 360x360
VAR_INPUT
    ITF_SPERRANTRIEBIN 	:	ITF_SPERRANTRIEB;
	ITF_RevSwitch_IN 	:	CtaSysIO.ITF_IO;
	ITF_Ready_IN 		:	CtaSysIO.ITF_IO;
	ITF_HandModul_IN 	:	CtaSysIO.ITF_IO;
END_VAR
    Frame (170,25 20x20)
        shows CtaSysConfig.visBOOL(visfbBOOLIn := ITF_SPERRANTRIEBIN.p_scInSperrAtRevisionSwitch_fbxEnable)
    Label (200,25 150x20), "Vorhanden"
    Frame (170,60 20x20)
        shows CtaSysConfig.visBOOL(visfbBOOLIn := ITF_SPERRANTRIEBIN.p_scInSperrAtRevisionSwitch_fbxInputMb)
    Label (200,60 150x20), "Signal via Modbus"
    Label (5,0 350x20), "Input Revisionsschalter"
    Label (5,95 350x20), "Input Bereitmeldung"
    Frame (170,120 20x20)
        shows CtaSysConfig.visBOOL(visfbBOOLIn := ITF_SPERRANTRIEBIN.p_scInSperrAtReady_fbxEnable)
    Label (200,120 150x20), "Vorhanden"
    Frame (170,155 20x20)
        shows CtaSysConfig.visBOOL(visfbBOOLIn := ITF_SPERRANTRIEBIN.p_scInSperrAtReady_fbxInputMb)
    Label (200,155 150x20), "Signal via Modbus"
    Label (5,195 350x20), "Input Handmodul"
    Frame (170,220 20x20)
        shows CtaSysConfig.visBOOL(visfbBOOLIn := ITF_SPERRANTRIEBIN.p_scInSperrAtHand_fbxEnable)
    Label (200,220 150x20), "Vorhanden"
    Frame (170,255 20x20)
        shows CtaSysConfig.visBOOL(visfbBOOLIn := ITF_SPERRANTRIEBIN.p_scInSperrAtHand_fbxInputMb)
    Label (200,255 150x20), "Signal via Modbus"
    Line (5,18) (354,18)
    Line (5,113) (354,113)
    Line (5,213) (354,213)
    Image (10,231 32x32), invisible if: ITF_HandModul_IN = 0, image: CtaVisSymbols.ImagePool.build
        OnMouseDown:  Dialog=SperrAntrieb_POPUP_IO_ITF, Parameters={ITF_IO_IN: ITF_HandModul_IN}, OpenModal=True, OpenCentered=True
    Image (10,35 32x32), invisible if: ITF_RevSwitch_IN = 0, image: CtaVisSymbols.ImagePool.build
        OnMouseDown:  Dialog=SperrAntrieb_POPUP_IO_ITF, Parameters={ITF_IO_IN: ITF_RevSwitch_IN}, OpenModal=True, OpenCentered=True
    Label (45,41 120x20), "IO- Konfiguration", invisible if: ITF_RevSwitch_IN = 0
    Image (10,130 32x32), invisible if: ITF_Ready_IN = 0, image: CtaVisSymbols.ImagePool.build
        OnMouseDown:  Dialog=SperrAntrieb_POPUP_IO_ITF, Parameters={ITF_IO_IN: ITF_Ready_IN}, OpenModal=True, OpenCentered=True
    Label (45,136 120x20), "IO- Konfiguration", invisible if: ITF_Ready_IN = 0
    Label (45,237 120x20), "IO- Konfiguration", invisible if: ITF_HandModul_IN = 0
END_VISUALIZATION

// 40 Visualizations/POPUP/PARAMETER/SperrAntrieb_IO/SperrAntrieb_ParameterIO1
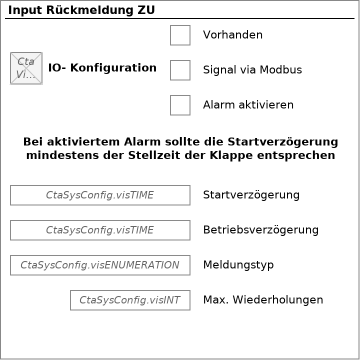
VISUALIZATION SperrAntrieb_ParameterIO1  // 360x360
VAR_INPUT
    ITF_SPERRANTRIEBIN 	:	ITF_SPERRANTRIEB;
	ITF_RückClosed_IN	:	CtaSysIO.ITF_IO;
END_VAR
    Label (5,0 350x20), "Input Rückmeldung ZU"
    Frame (170,25 20x20)
        shows CtaSysConfig.visBOOL(visfbBOOLIn := ITF_SPERRANTRIEBIN.p_scInSperrAtRükClosed_fbxEnable)
    Label (200,25 150x20), "Vorhanden"
    Frame (170,60 20x20)
        shows CtaSysConfig.visBOOL(visfbBOOLIn := ITF_SPERRANTRIEBIN.p_scInSperrAtRükClosed_fbxInputMb)
    Label (200,60 150x20), "Signal via Modbus"
    Frame (170,95 20x20)
        shows CtaSysConfig.visBOOL(visfbBOOLIn := ITF_SPERRANTRIEBIN.p_scInSperrAtRükClosed_fbxDoesAlarm)
    Label (200,95 150x20), "Alarm aktivieren"
    Frame (10,185 180x20)
        shows CtaSysConfig.visTIME(visfbTIMEIn := ITF_SPERRANTRIEBIN.p_scInSperrAtRükClosed_fbtDelayStart)
    Label (200,185 150x20), "Startverzögerung"
    Label (200,220 150x20), "Betriebsverzögerung"
    Frame (10,220 180x20)
        shows CtaSysConfig.visTIME(visfbTIMEIn := ITF_SPERRANTRIEBIN.p_scInSperrAtRükClosed_fbtDelayRun)
    Label (5,135 352x27), "Bei aktiviertem Alarm sollte die Startverzögerung mindestens der Stellzeit der Klappe entsprechen"
    Label (200,255 150x20), "Meldungstyp"
    Label (200,290 150x20), "Max. Wiederholungen"
    Line (5,18) (354,18)
    Frame (10,255 180x20), text list: 'CtaAppReport.txtLibAp99_2enTypeOfAck', text index: CtaSysConfig.fcGetEnumerationId(ITF_SPERRANTRIEBIN.p_scInSperrAtRükClosed_fbiTypeOfAck)
        shows CtaSysConfig.visENUMERATION(visfbENUIn := ITF_SPERRANTRIEBIN.p_scInSperrAtRükClosed_fbiTypeOfAck)
    Frame (70,290 120x20)
        shows CtaSysConfig.visINT(visfbINTIn := ITF_SPERRANTRIEBIN.p_scInSperrAtRükClosed_fbiMaxErrorRetryAllowed)
    Image (10,52 32x32), invisible if: ITF_RückClosed_IN = 0, image: CtaVisSymbols.ImagePool.build
        OnMouseDown:  Dialog=SperrAntrieb_POPUP_IO_ITF, Parameters={ITF_IO_IN: ITF_RückClosed_IN}, OpenModal=True, OpenCentered=True
    Label (45,58 120x20), "IO- Konfiguration", invisible if: ITF_RückClosed_IN = 0
END_VISUALIZATION

// 40 Visualizations/POPUP/PARAMETER/SperrAntrieb_IO/SperrAntrieb_ParameterIO
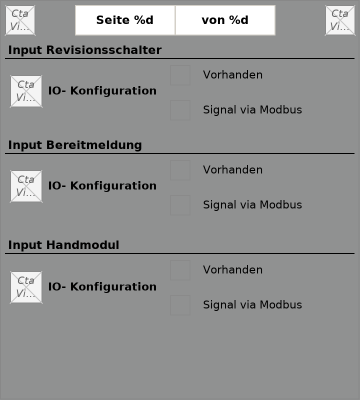
VISUALIZATION SperrAntrieb_ParameterIO  // 360x400
VAR_INPUT
    ITF_SPERRANTRIEBIN : ITF_SPERRANTRIEB;
END_VAR
VAR
    uiPage  :   UINT;
    uiMin   :   UINT    := 0;
    uiMax   :   UINT    := 4;
END_VAR
    Frame (0,40 360x360), frame switch variable: uiPage
        shows SperrAntrieb_ParameterIO0(ITF_SPERRANTRIEBIN := ITF_SPERRANTRIEBIN, ITF_RevSwitch_IN := ITF_SPERRANTRIEBIN.proRevisionSwitch_ITF, ITF_Ready_IN := ITF_SPERRANTRIEBIN.proActuatorReady_ITF, ITF_HandModul_IN := ITF_SPERRANTRIEBIN.proHandModul_ITF)
        shows SperrAntrieb_ParameterIO1(ITF_SPERRANTRIEBIN := ITF_SPERRANTRIEBIN, ITF_RückClosed_IN := ITF_SPERRANTRIEBIN.proIsClosed_ITF)
        shows SperrAntrieb_ParameterIO2(ITF_SPERRANTRIEBIN := ITF_SPERRANTRIEBIN, ITF_RückOffen_IN := ITF_SPERRANTRIEBIN.proIsOpen_ITF)
        shows SperrAntrieb_ParameterIO3(ITF_SPERRANTRIEBIN := ITF_SPERRANTRIEBIN, ITF_ActualPos_IN := ITF_SPERRANTRIEBIN.proActualPosition_ITF)
        shows SperrAntrieb_ParameterIO4(ITF_SPERRANTRIEBIN := ITF_SPERRANTRIEBIN, ITF_xOnAuf_IN := ITF_SPERRANTRIEBIN.proOnOpen_ITF, ITF_xOnZu_IN := ITF_SPERRANTRIEBIN.proOnClose_ITF, ITF_rOnY_IN := ITF_SPERRANTRIEBIN.proOnY_ITF)
    Image (325,5 30x30), invisible if: uiPage = uiMax, image: CtaVisSymbols.ImagePool.arrow-right_square
        OnMouseClick: execute {
            uiPage := uiPage + 1;
            IF uiPage >= uiMax THEN
                uiPage := uiMax;
            END_IF;
        }
    Image (5,5 30x30), invisible if: uiPage = uiMin, image: CtaVisSymbols.ImagePool.arrow-left_square
        OnMouseClick: execute {
            uiPage := uiPage - 1;
            IF uiPage <= uiMin THEN
                uiPage := uiMin;
            END_IF;
        }
    Textfield (175,5 100x30), "von %d", text variable: uiMax
    Textfield (75,5 100x30), "Seite %d", text variable: uiPage
END_VISUALIZATION

// 40 Visualizations/POPUP/PARAMETER/SperrAntrieb_IO/SperrAntrieb_ParameterIO2
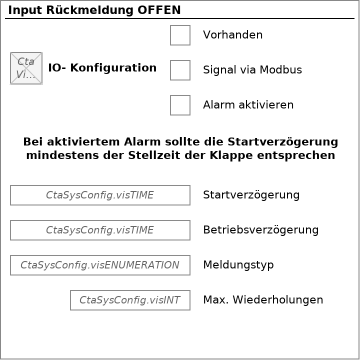
VISUALIZATION SperrAntrieb_ParameterIO2  // 360x360
VAR_INPUT
    ITF_SPERRANTRIEBIN 	:	ITF_SPERRANTRIEB;
	ITF_RückOffen_IN	:	CtaSysIO.ITF_IO;
END_VAR
    Label (5,0 350x20), "Input Rückmeldung OFFEN"
    Frame (170,25 20x20)
        shows CtaSysConfig.visBOOL(visfbBOOLIn := ITF_SPERRANTRIEBIN.p_scInSperrAtRükOpen_fbxEnable)
    Label (200,25 150x20), "Vorhanden"
    Frame (170,60 20x20)
        shows CtaSysConfig.visBOOL(visfbBOOLIn := ITF_SPERRANTRIEBIN.p_scInSperrAtRükOpen_fbxInputMb)
    Label (200,60 150x20), "Signal via Modbus"
    Frame (170,95 20x20)
        shows CtaSysConfig.visBOOL(visfbBOOLIn := ITF_SPERRANTRIEBIN.p_scInSperrAtRükOpen_fbxDoesAlarm)
    Label (200,95 150x20), "Alarm aktivieren"
    Frame (10,185 180x20)
        shows CtaSysConfig.visTIME(visfbTIMEIn := ITF_SPERRANTRIEBIN.p_scInSperrAtRükOpen_fbtDelayStart)
    Label (200,185 150x20), "Startverzögerung"
    Label (200,220 150x20), "Betriebsverzögerung"
    Frame (10,220 180x20)
        shows CtaSysConfig.visTIME(visfbTIMEIn := ITF_SPERRANTRIEBIN.p_scInSperrAtRükOpen_fbtDelayRun)
    Label (5,135 352x27), "Bei aktiviertem Alarm sollte die Startverzögerung mindestens der Stellzeit der Klappe entsprechen"
    Label (200,255 150x20), "Meldungstyp"
    Label (200,290 150x20), "Max. Wiederholungen"
    Line (5,18) (354,18)
    Frame (10,255 180x20), text list: 'CtaAppReport.txtLibAp99_2enTypeOfAck', text index: CtaSysConfig.fcGetEnumerationId(ITF_SPERRANTRIEBIN.p_scInSperrAtRükOpen_fbiTypeOfAck)
        shows CtaSysConfig.visENUMERATION(visfbENUIn := ITF_SPERRANTRIEBIN.p_scInSperrAtRükOpen_fbiTypeOfAck)
    Frame (70,290 120x20)
        shows CtaSysConfig.visINT(visfbINTIn := ITF_SPERRANTRIEBIN.p_scInSperrAtRükOpen_fbiMaxErrorRetryAllowed)
    Image (10,52 32x32), invisible if: ITF_RückOffen_IN = 0, image: CtaVisSymbols.ImagePool.build
        OnMouseDown:  Dialog=SperrAntrieb_POPUP_IO_ITF, Parameters={ITF_IO_IN: ITF_RückOffen_IN}, OpenModal=True, OpenCentered=True
    Label (45,58 120x20), "IO- Konfiguration", invisible if: ITF_RückOffen_IN = 0
END_VISUALIZATION

// 40 Visualizations/POPUP/PARAMETER/SperrAntrieb_IO/SperrAntrieb_ParameterIO3
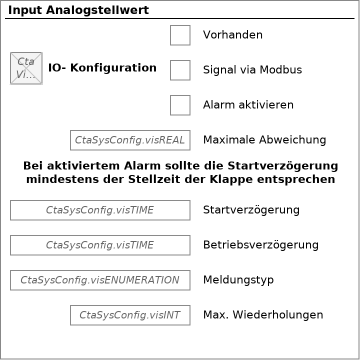
VISUALIZATION SperrAntrieb_ParameterIO3  // 360x360
VAR_INPUT
    ITF_SPERRANTRIEBIN 	:	ITF_SPERRANTRIEB;
	ITF_ActualPos_IN	:	CtaSysIO.ITF_IO;
END_VAR
    Label (5,0 350x20), "Input Analogstellwert"
    Frame (170,25 20x20)
        shows CtaSysConfig.visBOOL(visfbBOOLIn := ITF_SPERRANTRIEBIN.p_scInSperrAtActualPosition_fbxEnable)
    Label (200,25 150x20), "Vorhanden"
    Frame (170,60 20x20)
        shows CtaSysConfig.visBOOL(visfbBOOLIn := ITF_SPERRANTRIEBIN.p_scInSperrAtActualPosition_fbxInputMb)
    Label (200,60 150x20), "Signal via Modbus"
    Frame (170,95 20x20)
        shows CtaSysConfig.visBOOL(visfbBOOLIn := ITF_SPERRANTRIEBIN.p_scInSperrAtActualPosition_fbxDoesAlarm)
    Label (200,95 150x20), "Alarm aktivieren"
    Frame (10,200 180x20)
        shows CtaSysConfig.visTIME(visfbTIMEIn := ITF_SPERRANTRIEBIN.p_scInSperrAtActualPosition_fbtDelayStart)
    Label (200,200 150x20), "Startverzögerung"
    Label (200,235 150x20), "Betriebsverzögerung"
    Frame (10,235 180x20)
        shows CtaSysConfig.visTIME(visfbTIMEIn := ITF_SPERRANTRIEBIN.p_scInSperrAtActualPosition_fbtDelayRun)
    Frame (70,130 120x20)
        shows CtaSysConfig.visREAL(visfbREALIn := ITF_SPERRANTRIEBIN.p_scInSperrAtActualPosition_fbrMaxDiff, stPhysikalischeEinheit := '%')
    Label (200,130 150x20), "Maximale Abweichung"
    Label (5,159 352x27), "Bei aktiviertem Alarm sollte die Startverzögerung mindestens der Stellzeit der Klappe entsprechen"
    Label (200,270 150x20), "Meldungstyp"
    Label (200,305 150x20), "Max. Wiederholungen"
    Line (5,18) (354,18)
    Frame (10,270 180x20), text list: 'CtaAppReport.txtLibAp99_2enTypeOfAck', text index: CtaSysConfig.fcGetEnumerationId(ITF_SPERRANTRIEBIN.p_scInSperrAtActualPosition_fbiTypeOfAck)
        shows CtaSysConfig.visENUMERATION(visfbENUIn := ITF_SPERRANTRIEBIN.p_scInSperrAtActualPosition_fbiTypeOfAck)
    Frame (70,305 120x20)
        shows CtaSysConfig.visINT(visfbINTIn := ITF_SPERRANTRIEBIN.p_scInSperrAtActualPosition_fbiMaxErrorRetryAllowed)
    Image (10,52 32x32), invisible if: ITF_ActualPos_IN = 0, image: CtaVisSymbols.ImagePool.build
        OnMouseDown:  Dialog=SperrAntrieb_POPUP_IO_ITF, Parameters={ITF_IO_IN: ITF_ActualPos_IN}, OpenModal=True, OpenCentered=True
    Label (45,58 120x20), "IO- Konfiguration", invisible if: ITF_ActualPos_IN = 0
END_VISUALIZATION

// 40 Visualizations/POPUP/PARAMETER/SperrAntrieb_InfluxDb/SperrAntrieb_ParameterInfluxDb
